//     Term 27 (APS4322-7000)/Term 28 (APS4322-5000)/FB Inputs/I{0..8 step 2} Y-Field <-> Data Pointer/HallSensorFieldsXYZ[{121..133 step 3}]  (5 links)
//     Term 27 (APS4322-7000)/Term 28 (APS4322-5000)/FB Inputs/I{0..8 step 2} Z-Field <-> Data Pointer/HallSensorFieldsXYZ[{122..134 step 3}]  (5 links)
//     Term 27 (APS4322-7000)/Term 28 (APS4322-5000)/FB Inputs/J{1..9 step 2} X-Field <-> Data Pointer/HallSensorFieldsXYZ[{135..147 step 3}]  (5 links)
//     Term 27 (APS4322-7000)/Term 28 (APS4322-5000)/FB Inputs/J{1..9 step 2} Y-Field <-> Data Pointer/HallSensorFieldsXYZ[{136..148 step 3}]  (5 links)
//     Term 27 (APS4322-7000)/Term 28 (APS4322-5000)/FB Inputs/J{1..9 step 2} Z-Field <-> Data Pointer/HallSensorFieldsXYZ[{137..149 step 3}]  (5 links)
//     Term 27 (APS4322-7000)/Term 28 (APS4322-5000)/FB Inputs/Status <-> Data Pointer/FeedbackStatus
//   Device 2 (EtherCAT) <-> TcCOM Objects/XPlanar/Part1/Tile3
//     Term 17 (APS4322-7000)/APS Comm Inputs/CommStatusWord <-> Data Pointer/MoverCommStatusWord
//     Term 17 (APS4322-7000)/APS Comm Inputs/Data {1..4} <-> Data Pointer/MoverCommDataIn[{0..3}]  (4 links)
//     Term 17 (APS4322-7000)/APS Comm Outputs/CommControlWord <-> Data Pointer/MoverCommControlWord
//     Term 17 (APS4322-7000)/APS Comm Outputs/Data 1 <-> Data Pointer/MoverCommDataOut
//     Term 17 (APS4322-7000)/APS Diagdata/DC Link Voltage <-> Data Pointer/DcLinkVoltage
//     Term 17 (APS4322-7000)/APS Diagdata/Power supply current <-> Data Pointer/PowerSupplyCurrent
//     Term 17 (APS4322-7000)/APS Inputs/StatusWord <-> Data Pointer/PowerUnitStatusWord
//     Term 17 (APS4322-7000)/APS Outputs/ControlWord <-> Data Pointer/PowerUnitControlWord
//     Term 17 (APS4322-7000)/APS Outputs/Current D 0X0 <-> Data Pointer/DCurrentSetPoints[0]
//     Term 17 (APS4322-7000)/APS Outputs/Current D 0X1 <-> Data Pointer/DCurrentSetPoints[1]
//     Term 17 (APS4322-7000)/APS Outputs/Current D 0X2 <-> Data Pointer/DCurrentSetPoints[2]
//     Term 17 (APS4322-7000)/APS Outputs/Current D 1X0 <-> Data Pointer/DCurrentSetPoints[6]
//     Term 17 (APS4322-7000)/APS Outputs/Current D 1X1 <-> Data Pointer/DCurrentSetPoints[7]
//     Term 17 (APS4322-7000)/APS Outputs/Current D 1X2 <-> Data Pointer/DCurrentSetPoints[8]
//     Term 17 (APS4322-7000)/APS Outputs/Current D 2X0 <-> Data Pointer/DCurrentSetPoints[12]
//     Term 17 (APS4322-7000)/APS Outputs/Current D 2X1 <-> Data Pointer/DCurrentSetPoints[13]
//     Term 17 (APS4322-7000)/APS Outputs/Current D 2X2 <-> Data Pointer/DCurrentSetPoints[14]
//     Term 17 (APS4322-7000)/APS Outputs/Current D 3X0 <-> Data Pointer/DCurrentSetPoints[18]
//     Term 17 (APS4322-7000)/APS Outputs/Current D 3X1 <-> Data Pointer/DCurrentSetPoints[19]
//     Term 17 (APS4322-7000)/APS Outputs/Current D 3X2 <-> Data Pointer/DCurrentSetPoints[20]
//     Term 17 (APS4322-7000)/APS Outputs/Current D 0Y0 <-> Data Pointer/DCurrentSetPoints[3]
//     Term 17 (APS4322-7000)/APS Outputs/Current D 0Y1 <-> Data Pointer/DCurrentSetPoints[4]
//     Term 17 (APS4322-7000)/APS Outputs/Current D 0Y2 <-> Data Pointer/DCurrentSetPoints[5]
//     Term 17 (APS4322-7000)/APS Outputs/Current D 1Y0 <-> Data Pointer/DCurrentSetPoints[9]
//     Term 17 (APS4322-7000)/APS Outputs/Current D 1Y1 <-> Data Pointer/DCurrentSetPoints[10]
//     Term 17 (APS4322-7000)/APS Outputs/Current D 1Y2 <-> Data Pointer/DCurrentSetPoints[11]
//     Term 17 (APS4322-7000)/APS Outputs/Current D 2Y0 <-> Data Pointer/DCurrentSetPoints[15]
//     Term 17 (APS4322-7000)/APS Outputs/Current D 2Y1 <-> Data Pointer/DCurrentSetPoints[16]
//     Term 17 (APS4322-7000)/APS Outputs/Current D 2Y2 <-> Data Pointer/DCurrentSetPoints[17]
//     Term 17 (APS4322-7000)/APS Outputs/Current D 3Y0 <-> Data Pointer/DCurrentSetPoints[21]
//     Term 17 (APS4322-7000)/APS Outputs/Current D 3Y1 <-> Data Pointer/DCurrentSetPoints[22]
//     Term 17 (APS4322-7000)/APS Outputs/Current D 3Y2 <-> Data Pointer/DCurrentSetPoints[23]
//     Term 17 (APS4322-7000)/APS Outputs/Current Q 0X0 <-> Data Pointer/QCurrentSetPoints[0]
//     Term 17 (APS4322-7000)/APS Outputs/Current Q 0X1 <-> Data Pointer/QCurrentSetPoints[1]
//     Term 17 (APS4322-7000)/APS Outputs/Current Q 0X2 <-> Data Pointer/QCurrentSetPoints[2]
//     Term 17 (APS4322-7000)/APS Outputs/Current Q 1X0 <-> Data Pointer/QCurrentSetPoints[6]
//     Term 17 (APS4322-7000)/APS Outputs/Current Q 1X1 <-> Data Pointer/QCurrentSetPoints[7]
//     Term 17 (APS4322-7000)/APS Outputs/Current Q 1X2 <-> Data Pointer/QCurrentSetPoints[8]
//     Term 17 (APS4322-7000)/APS Outputs/Current Q 2X0 <-> Data Pointer/QCurrentSetPoints[12]
//     Term 17 (APS4322-7000)/APS Outputs/Current Q 2X1 <-> Data Pointer/QCurrentSetPoints[13]
//     Term 17 (APS4322-7000)/APS Outputs/Current Q 2X2 <-> Data Pointer/QCurrentSetPoints[14]
//     Term 17 (APS4322-7000)/APS Outputs/Current Q 3X0 <-> Data Pointer/QCurrentSetPoints[18]
//     Term 17 (APS4322-7000)/APS Outputs/Current Q 3X1 <-> Data Pointer/QCurrentSetPoints[19]
//     Term 17 (APS4322-7000)/APS Outputs/Current Q 3X2 <-> Data Pointer/QCurrentSetPoints[20]
//     Term 17 (APS4322-7000)/APS Outputs/Current Q 0Y0 <-> Data Pointer/QCurrentSetPoints[3]
//     Term 17 (APS4322-7000)/APS Outputs/Current Q 0Y1 <-> Data Pointer/QCurrentSetPoints[4]
//     Term 17 (APS4322-7000)/APS Outputs/Current Q 0Y2 <-> Data Pointer/QCurrentSetPoints[5]
//     Term 17 (APS4322-7000)/APS Outputs/Current Q 1Y0 <-> Data Pointer/QCurrentSetPoints[9]
//     Term 17 (APS4322-7000)/APS Outputs/Current Q 1Y1 <-> Data Pointer/QCurrentSetPoints[10]
//     Term 17 (APS4322-7000)/APS Outputs/Current Q 1Y2 <-> Data Pointer/QCurrentSetPoints[11]
//     Term 17 (APS4322-7000)/APS Outputs/Current Q 2Y0 <-> Data Pointer/QCurrentSetPoints[15]
//     Term 17 (APS4322-7000)/APS Outputs/Current Q 2Y1 <-> Data Pointer/QCurrentSetPoints[16]
//     Term 17 (APS4322-7000)/APS Outputs/Current Q 2Y2 <-> Data Pointer/QCurrentSetPoints[17]
//     Term 17 (APS4322-7000)/APS Outputs/Current Q 3Y0 <-> Data Pointer/QCurrentSetPoints[21]
//     Term 17 (APS4322-7000)/APS Outputs/Current Q 3Y1 <-> Data Pointer/QCurrentSetPoints[22]
//     Term 17 (APS4322-7000)/APS Outputs/Current Q 3Y2 <-> Data Pointer/QCurrentSetPoints[23]
//     Term 17 (APS4322-7000)/APS Outputs/PhiE 0X0 <-> Data Pointer/PhiSetPoints[0]
//     Term 17 (APS4322-7000)/APS Outputs/PhiE 0X1 <-> Data Pointer/PhiSetPoints[1]
//     Term 17 (APS4322-7000)/APS Outputs/PhiE 0X2 <-> Data Pointer/PhiSetPoints[2]
//     Term 17 (APS4322-7000)/APS Outputs/PhiE 1X0 <-> Data Pointer/PhiSetPoints[6]
//     Term 17 (APS4322-7000)/APS Outputs/PhiE 1X1 <-> Data Pointer/PhiSetPoints[7]
//     Term 17 (APS4322-7000)/APS Outputs/PhiE 1X2 <-> Data Pointer/PhiSetPoints[8]
//     Term 17 (APS4322-7000)/APS Outputs/PhiE 2X0 <-> Data Pointer/PhiSetPoints[12]
//     Term 17 (APS4322-7000)/APS Outputs/PhiE 2X1 <-> Data Pointer/PhiSetPoints[13]
//     Term 17 (APS4322-7000)/APS Outputs/PhiE 2X2 <-> Data Pointer/PhiSetPoints[14]
//     Term 17 (APS4322-7000)/APS Outputs/PhiE 3X0 <-> Data Pointer/PhiSetPoints[18]
//     Term 17 (APS4322-7000)/APS Outputs/PhiE 3X1 <-> Data Pointer/PhiSetPoints[19]
//     Term 17 (APS4322-7000)/APS Outputs/PhiE 3X2 <-> Data Pointer/PhiSetPoints[20]
//     Term 17 (APS4322-7000)/APS Outputs/PhiE 0Y0 <-> Data Pointer/PhiSetPoints[3]
//     Term 17 (APS4322-7000)/APS Outputs/PhiE 0Y1 <-> Data Pointer/PhiSetPoints[4]
//     Term 17 (APS4322-7000)/APS Outputs/PhiE 0Y2 <-> Data Pointer/PhiSetPoints[5]
//     Term 17 (APS4322-7000)/APS Outputs/PhiE 1Y0 <-> Data Pointer/PhiSetPoints[9]
//     Term 17 (APS4322-7000)/APS Outputs/PhiE 1Y1 <-> Data Pointer/PhiSetPoints[10]
//     Term 17 (APS4322-7000)/APS Outputs/PhiE 1Y2 <-> Data Pointer/PhiSetPoints[11]
//     Term 17 (APS4322-7000)/APS Outputs/PhiE 2Y0 <-> Data Pointer/PhiSetPoints[15]
//     Term 17 (APS4322-7000)/APS Outputs/PhiE 2Y1 <-> Data Pointer/PhiSetPoints[16]
//     Term 17 (APS4322-7000)/APS Outputs/PhiE 2Y2 <-> Data Pointer/PhiSetPoints[17]
//     Term 17 (APS4322-7000)/APS Outputs/PhiE 3Y0 <-> Data Pointer/PhiSetPoints[21]
//     Term 17 (APS4322-7000)/APS Outputs/PhiE 3Y1 <-> Data Pointer/PhiSetPoints[22]
//     Term 17 (APS4322-7000)/APS Outputs/PhiE 3Y2 <-> Data Pointer/PhiSetPoints[23]
//     Term 17 (APS4322-7000)/Term 18 (APS4322-5000)/FB Inputs/A{0..8 step 2} X-Field <-> Data Pointer/HallSensorFieldsXYZ[{0..12 step 3}]  (5 links)
//     Term 17 (APS4322-7000)/Term 18 (APS4322-5000)/FB Inputs/A{0..8 step 2} Y-Field <-> Data Pointer/HallSensorFieldsXYZ[{1..13 step 3}]  (5 links)
//     Term 17 (APS4322-7000)/Term 18 (APS4322-5000)/FB Inputs/A{0..8 step 2} Z-Field <-> Data Pointer/HallSensorFieldsXYZ[{2..14 step 3}]  (5 links)
//     Term 17 (APS4322-7000)/Term 18 (APS4322-5000)/FB Inputs/B{1..9 step 2} X-Field <-> Data Pointer/HallSensorFieldsXYZ[{15..27 step 3}]  (5 links)
//     Term 17 (APS4322-7000)/Term 18 (APS4322-5000)/FB Inputs/B{1..9 step 2} Y-Field <-> Data Pointer/HallSensorFieldsXYZ[{16..28 step 3}]  (5 links)
//     Term 17 (APS4322-7000)/Term 18 (APS4322-5000)/FB Inputs/B{1..9 step 2} Z-Field <-> Data Pointer/HallSensorFieldsXYZ[{17..29 step 3}]  (5 links)
//     Term 17 (APS4322-7000)/Term 18 (APS4322-5000)/FB Inputs/C{0..8 step 2} X-Field <-> Data Pointer/HallSensorFieldsXYZ[{30..42 step 3}]  (5 links)
//     Term 17 (APS4322-7000)/Term 18 (APS4322-5000)/FB Inputs/C{0..8 step 2} Y-Field <-> Data Pointer/HallSensorFieldsXYZ[{31..43 step 3}]  (5 links)
//     Term 17 (APS4322-7000)/Term 18 (APS4322-5000)/FB Inputs/C{0..8 step 2} Z-Field <-> Data Pointer/HallSensorFieldsXYZ[{32..44 step 3}]  (5 links)
//     Term 17 (APS4322-7000)/Term 18 (APS4322-5000)/FB Inputs/D{1..9 step 2} X-Field <-> Data Pointer/HallSensorFieldsXYZ[{45..57 step 3}]  (5 links)
//     Term 17 (APS4322-7000)/Term 18 (APS4322-5000)/FB Inputs/D{1..9 step 2} Y-Field <-> Data Pointer/HallSensorFieldsXYZ[{46..58 step 3}]  (5 links)
//     Term 17 (APS4322-7000)/Term 18 (APS4322-5000)/FB Inputs/D{1..9 step 2} Z-Field <-> Data Pointer/HallSensorFieldsXYZ[{47..59 step 3}]  (5 links)
//     Term 17 (APS4322-7000)/Term 18 (APS4322-5000)/FB Inputs/E{0..8 step 2} X-Field <-> Data Pointer/HallSensorFieldsXYZ[{60..72 step 3}]  (5 links)
//     Term 17 (APS4322-7000)/Term 18 (APS4322-5000)/FB Inputs/E{0..8 step 2} Y-Field <-> Data Pointer/HallSensorFieldsXYZ[{61..73 step 3}]  (5 links)
//     Term 17 (APS4322-7000)/Term 18 (APS4322-5000)/FB Inputs/E{0..8 step 2} Z-Field <-> Data Pointer/HallSensorFieldsXYZ[{62..74 step 3}]  (5 links)
//     Term 17 (APS4322-7000)/Term 18 (APS4322-5000)/FB Inputs/F{1..9 step 2} X-Field <-> Data Pointer/HallSensorFieldsXYZ[{75..87 step 3}]  (5 links)
//     Term 17 (APS4322-7000)/Term 18 (APS4322-5000)/FB Inputs/F{1..9 step 2} Y-Field <-> Data Pointer/HallSensorFieldsXYZ[{76..88 step 3}]  (5 links)
//     Term 17 (APS4322-7000)/Term 18 (APS4322-5000)/FB Inputs/F{1..9 step 2} Z-Field <-> Data Pointer/HallSensorFieldsXYZ[{77..89 step 3}]  (5 links)
//     Term 17 (APS4322-7000)/Term 18 (APS4322-5000)/FB Inputs/G{0..8 step 2} X-Field <-> Data Pointer/HallSensorFieldsXYZ[{90..102 step 3}]  (5 links)
//     Term 17 (APS4322-7000)/Term 18 (APS4322-5000)/FB Inputs/G{0..8 step 2} Y-Field <-> Data Pointer/HallSensorFieldsXYZ[{91..103 step 3}]  (5 links)
//     Term 17 (APS4322-7000)/Term 18 (APS4322-5000)/FB Inputs/G{0..8 step 2} Z-Field <-> Data Pointer/HallSensorFieldsXYZ[{92..104 step 3}]  (5 links)
//     Term 17 (APS4322-7000)/Term 18 (APS4322-5000)/FB Inputs/H{1..9 step 2} X-Field <-> Data Pointer/HallSensorFieldsXYZ[{105..117 step 3}]  (5 links)
//     Term 17 (APS4322-7000)/Term 18 (APS4322-5000)/FB Inputs/H{1..9 step 2} Y-Field <-> Data Pointer/HallSensorFieldsXYZ[{106..118 step 3}]  (5 links)
//     Term 17 (APS4322-7000)/Term 18 (APS4322-5000)/FB Inputs/H{1..9 step 2} Z-Field <-> Data Pointer/HallSensorFieldsXYZ[{107..119 step 3}]  (5 links)
//     Term 17 (APS4322-7000)/Term 18 (APS4322-5000)/FB Inputs/I{0..8 step 2} X-Field <-> Data Pointer/HallSensorFieldsXYZ[{120..132 step 3}]  (5 links)
//     Term 17 (APS4322-7000)/Term 18 (APS4322-5000)/FB Inputs/I{0..8 step 2} Y-Field <-> Data Pointer/HallSensorFieldsXYZ[{121..133 step 3}]  (5 links)
//     Term 17 (APS4322-7000)/Term 18 (APS4322-5000)/FB Inputs/I{0..8 step 2} Z-Field <-> Data Pointer/HallSensorFieldsXYZ[{122..134 step 3}]  (5 links)
//     Term 17 (APS4322-7000)/Term 18 (APS4322-5000)/FB Inputs/J{1..9 step 2} X-Field <-> Data Pointer/HallSensorFieldsXYZ[{135..147 step 3}]  (5 links)
//     Term 17 (APS4322-7000)/Term 18 (APS4322-5000)/FB Inputs/J{1..9 step 2} Y-Field <-> Data Pointer/HallSensorFieldsXYZ[{136..148 step 3}]  (5 links)
//     Term 17 (APS4322-7000)/Term 18 (APS4322-5000)/FB Inputs/J{1..9 step 2} Z-Field <-> Data Pointer/HallSensorFieldsXYZ[{137..149 step 3}]  (5 links)
//     Term 17 (APS4322-7000)/Term 18 (APS4322-5000)/FB Inputs/Status <-> Data Pointer/FeedbackStatus
//   Device 2 (EtherCAT) <-> TcCOM Objects/XPlanar/Part1/Tile4
//     Term 19 (APS4322-7000)/APS Comm Inputs/CommStatusWord <-> Data Pointer/MoverCommStatusWord
//     Term 19 (APS4322-7000)/APS Comm Inputs/Data {1..4} <-> Data Pointer/MoverCommDataIn[{0..3}]  (4 links)
//     Term 19 (APS4322-7000)/APS Comm Outputs/CommControlWord <-> Data Pointer/MoverCommControlWord
//     Term 19 (APS4322-7000)/APS Comm Outputs/Data 1 <-> Data Pointer/MoverCommDataOut
//     Term 19 (APS4322-7000)/APS Diagdata/DC Link Voltage <-> Data Pointer/DcLinkVoltage
//     Term 19 (APS4322-7000)/APS Diagdata/Power supply current <-> Data Pointer/PowerSupplyCurrent
//     Term 19 (APS4322-7000)/APS Inputs/StatusWord <-> Data Pointer/PowerUnitStatusWord
//     Term 19 (APS4322-7000)/APS Outputs/ControlWord <-> Data Pointer/PowerUnitControlWord
//     Term 19 (APS4322-7000)/APS Outputs/Current D 0X0 <-> Data Pointer/DCurrentSetPoints[0]
//     Term 19 (APS4322-7000)/APS Outputs/Current D 0X1 <-> Data Pointer/DCurrentSetPoints[1]
//     Term 19 (APS4322-7000)/APS Outputs/Current D 0X2 <-> Data Pointer/DCurrentSetPoints[2]
//     Term 19 (APS4322-7000)/APS Outputs/Current D 1X0 <-> Data Pointer/DCurrentSetPoints[6]
//     Term 19 (APS4322-7000)/APS Outputs/Current D 1X1 <-> Data Pointer/DCurrentSetPoints[7]
//     Term 19 (APS4322-7000)/APS Outputs/Current D 1X2 <-> Data Pointer/DCurrentSetPoints[8]
//     Term 19 (APS4322-7000)/APS Outputs/Current D 2X0 <-> Data Pointer/DCurrentSetPoints[12]
//     Term 19 (APS4322-7000)/APS Outputs/Current D 2X1 <-> Data Pointer/DCurrentSetPoints[13]
//     Term 19 (APS4322-7000)/APS Outputs/Current D 2X2 <-> Data Pointer/DCurrentSetPoints[14]
//     Term 19 (APS4322-7000)/APS Outputs/Current D 3X0 <-> Data Pointer/DCurrentSetPoints[18]
//     Term 19 (APS4322-7000)/APS Outputs/Current D 3X1 <-> Data Pointer/DCurrentSetPoints[19]
//     Term 19 (APS4322-7000)/APS Outputs/Current D 3X2 <-> Data Pointer/DCurrentSetPoints[20]
//     Term 19 (APS4322-7000)/APS Outputs/Current D 0Y0 <-> Data Pointer/DCurrentSetPoints[3]
//     Term 19 (APS4322-7000)/APS Outputs/Current D 0Y1 <-> Data Pointer/DCurrentSetPoints[4]
//     Term 19 (APS4322-7000)/APS Outputs/Current D 0Y2 <-> Data Pointer/DCurrentSetPoints[5]
//     Term 19 (APS4322-7000)/APS Outputs/Current D 1Y0 <-> Data Pointer/DCurrentSetPoints[9]
//     Term 19 (APS4322-7000)/APS Outputs/Current D 1Y1 <-> Data Pointer/DCurrentSetPoints[10]
//     Term 19 (APS4322-7000)/APS Outputs/Current D 1Y2 <-> Data Pointer/DCurrentSetPoints[11]
//     Term 19 (APS4322-7000)/APS Outputs/Current D 2Y0 <-> Data Pointer/DCurrentSetPoints[15]
//     Term 19 (APS4322-7000)/APS Outputs/Current D 2Y1 <-> Data Pointer/DCurrentSetPoints[16]
//     Term 19 (APS4322-7000)/APS Outputs/Current D 2Y2 <-> Data Pointer/DCurrentSetPoints[17]
//     Term 19 (APS4322-7000)/APS Outputs/Current D 3Y0 <-> Data Pointer/DCurrentSetPoints[21]
//     Term 19 (APS4322-7000)/APS Outputs/Current D 3Y1 <-> Data Pointer/DCurrentSetPoints[22]
//     Term 19 (APS4322-7000)/APS Outputs/Current D 3Y2 <-> Data Pointer/DCurrentSetPoints[23]
//     Term 19 (APS4322-7000)/APS Outputs/Current Q 0X0 <-> Data Pointer/QCurrentSetPoints[0]
//     Term 19 (APS4322-7000)/APS Outputs/Current Q 0X1 <-> Data Pointer/QCurrentSetPoints[1]
//     Term 19 (APS4322-7000)/APS Outputs/Current Q 0X2 <-> Data Pointer/QCurrentSetPoints[2]
//     Term 19 (APS4322-7000)/APS Outputs/Current Q 1X0 <-> Data Pointer/QCurrentSetPoints[6]
//     Term 19 (APS4322-7000)/APS Outputs/Current Q 1X1 <-> Data Pointer/QCurrentSetPoints[7]
//     Term 19 (APS4322-7000)/APS Outputs/Current Q 1X2 <-> Data Pointer/QCurrentSetPoints[8]
//     Term 19 (APS4322-7000)/APS Outputs/Current Q 2X0 <-> Data Pointer/QCurrentSetPoints[12]
//     Term 19 (APS4322-7000)/APS Outputs/Current Q 2X1 <-> Data Pointer/QCurrentSetPoints[13]
//     Term 19 (APS4322-7000)/APS Outputs/Current Q 2X2 <-> Data Pointer/QCurrentSetPoints[14]
//     Term 19 (APS4322-7000)/APS Outputs/Current Q 3X0 <-> Data Pointer/QCurrentSetPoints[18]
//     Term 19 (APS4322-7000)/APS Outputs/Current Q 3X1 <-> Data Pointer/QCurrentSetPoints[19]
//     Term 19 (APS4322-7000)/APS Outputs/Current Q 3X2 <-> Data Pointer/QCurrentSetPoints[20]
//     Term 19 (APS4322-7000)/APS Outputs/Current Q 0Y0 <-> Data Pointer/QCurrentSetPoints[3]
//     Term 19 (APS4322-7000)/APS Outputs/Current Q 0Y1 <-> Data Pointer/QCurrentSetPoints[4]
//     Term 19 (APS4322-7000)/APS Outputs/Current Q 0Y2 <-> Data Pointer/QCurrentSetPoints[5]
//     Term 19 (APS4322-7000)/APS Outputs/Current Q 1Y0 <-> Data Pointer/QCurrentSetPoints[9]
//     Term 19 (APS4322-7000)/APS Outputs/Current Q 1Y1 <-> Data Pointer/QCurrentSetPoints[10]
//     Term 19 (APS4322-7000)/APS Outputs/Current Q 1Y2 <-> Data Pointer/QCurrentSetPoints[11]
//     Term 19 (APS4322-7000)/APS Outputs/Current Q 2Y0 <-> Data Pointer/QCurrentSetPoints[15]
//     Term 19 (APS4322-7000)/APS Outputs/Current Q 2Y1 <-> Data Pointer/QCurrentSetPoints[16]
//     Term 19 (APS4322-7000)/APS Outputs/Current Q 2Y2 <-> Data Pointer/QCurrentSetPoints[17]
//     Term 19 (APS4322-7000)/APS Outputs/Current Q 3Y0 <-> Data Pointer/QCurrentSetPoints[21]
//     Term 19 (APS4322-7000)/APS Outputs/Current Q 3Y1 <-> Data Pointer/QCurrentSetPoints[22]
//     Term 19 (APS4322-7000)/APS Outputs/Current Q 3Y2 <-> Data Pointer/QCurrentSetPoints[23]
//     Term 19 (APS4322-7000)/APS Outputs/PhiE 0X0 <-> Data Pointer/PhiSetPoints[0]
//     Term 19 (APS4322-7000)/APS Outputs/PhiE 0X1 <-> Data Pointer/PhiSetPoints[1]
//     Term 19 (APS4322-7000)/APS Outputs/PhiE 0X2 <-> Data Pointer/PhiSetPoints[2]
//     Term 19 (APS4322-7000)/APS Outputs/PhiE 1X0 <-> Data Pointer/PhiSetPoints[6]
//     Term 19 (APS4322-7000)/APS Outputs/PhiE 1X1 <-> Data Pointer/PhiSetPoints[7]
//     Term 19 (APS4322-7000)/APS Outputs/PhiE 1X2 <-> Data Pointer/PhiSetPoints[8]
//     Term 19 (APS4322-7000)/APS Outputs/PhiE 2X0 <-> Data Pointer/PhiSetPoints[12]
//     Term 19 (APS4322-7000)/APS Outputs/PhiE 2X1 <-> Data Pointer/PhiSetPoints[13]
//     Term 19 (APS4322-7000)/APS Outputs/PhiE 2X2 <-> Data Pointer/PhiSetPoints[14]
//     Term 19 (APS4322-7000)/APS Outputs/PhiE 3X0 <-> Data Pointer/PhiSetPoints[18]
//     Term 19 (APS4322-7000)/APS Outputs/PhiE 3X1 <-> Data Pointer/PhiSetPoints[19]
//     Term 19 (APS4322-7000)/APS Outputs/PhiE 3X2 <-> Data Pointer/PhiSetPoints[20]
//     Term 19 (APS4322-7000)/APS Outputs/PhiE 0Y0 <-> Data Pointer/PhiSetPoints[3]
//     Term 19 (APS4322-7000)/APS Outputs/PhiE 0Y1 <-> Data Pointer/PhiSetPoints[4]
//     Term 19 (APS4322-7000)/APS Outputs/PhiE 0Y2 <-> Data Pointer/PhiSetPoints[5]
//     Term 19 (APS4322-7000)/APS Outputs/PhiE 1Y0 <-> Data Pointer/PhiSetPoints[9]
//     Term 19 (APS4322-7000)/APS Outputs/PhiE 1Y1 <-> Data Pointer/PhiSetPoints[10]
//     Term 19 (APS4322-7000)/APS Outputs/PhiE 1Y2 <-> Data Pointer/PhiSetPoints[11]
//     Term 19 (APS4322-7000)/APS Outputs/PhiE 2Y0 <-> Data Pointer/PhiSetPoints[15]
//     Term 19 (APS4322-7000)/APS Outputs/PhiE 2Y1 <-> Data Pointer/PhiSetPoints[16]
//     Term 19 (APS4322-7000)/APS Outputs/PhiE 2Y2 <-> Data Pointer/PhiSetPoints[17]
//     Term 19 (APS4322-7000)/APS Outputs/PhiE 3Y0 <-> Data Pointer/PhiSetPoints[21]
//     Term 19 (APS4322-7000)/APS Outputs/PhiE 3Y1 <-> Data Pointer/PhiSetPoints[22]
//     Term 19 (APS4322-7000)/APS Outputs/PhiE 3Y2 <-> Data Pointer/PhiSetPoints[23]
//     Term 19 (APS4322-7000)/Term 20 (APS4322-5000)/FB Inputs/A{0..8 step 2} X-Field <-> Data Pointer/HallSensorFieldsXYZ[{0..12 step 3}]  (5 links)
//     Term 19 (APS4322-7000)/Term 20 (APS4322-5000)/FB Inputs/A{0..8 step 2} Y-Field <-> Data Pointer/HallSensorFieldsXYZ[{1..13 step 3}]  (5 links)
//     Term 19 (APS4322-7000)/Term 20 (APS4322-5000)/FB Inputs/A{0..8 step 2} Z-Field <-> Data Pointer/HallSensorFieldsXYZ[{2..14 step 3}]  (5 links)
//     Term 19 (APS4322-7000)/Term 20 (APS4322-5000)/FB Inputs/B{1..9 step 2} X-Field <-> Data Pointer/HallSensorFieldsXYZ[{15..27 step 3}]  (5 links)
//     Term 19 (APS4322-7000)/Term 20 (APS4322-5000)/FB Inputs/B{1..9 step 2} Y-Field <-> Data Pointer/HallSensorFieldsXYZ[{16..28 step 3}]  (5 links)
//     Term 19 (APS4322-7000)/Term 20 (APS4322-5000)/FB Inputs/B{1..9 step 2} Z-Field <-> Data Pointer/HallSensorFieldsXYZ[{17..29 step 3}]  (5 links)
//     Term 19 (APS4322-7000)/Term 20 (APS4322-5000)/FB Inputs/C{0..8 step 2} X-Field <-> Data Pointer/HallSensorFieldsXYZ[{30..42 step 3}]  (5 links)
//     Term 19 (APS4322-7000)/Term 20 (APS4322-5000)/FB Inputs/C{0..8 step 2} Y-Field <-> Data Pointer/HallSensorFieldsXYZ[{31..43 step 3}]  (5 links)
//     Term 19 (APS4322-7000)/Term 20 (APS4322-5000)/FB Inputs/C{0..8 step 2} Z-Field <-> Data Pointer/HallSensorFieldsXYZ[{32..44 step 3}]  (5 links)
//     Term 19 (APS4322-7000)/Term 20 (APS4322-5000)/FB Inputs/D{1..9 step 2} X-Field <-> Data Pointer/HallSensorFieldsXYZ[{45..57 step 3}]  (5 links)
//     Term 19 (APS4322-7000)/Term 20 (APS4322-5000)/FB Inputs/D{1..9 step 2} Y-Field <-> Data Pointer/HallSensorFieldsXYZ[{46..58 step 3}]  (5 links)
//     Term 19 (APS4322-7000)/Term 20 (APS4322-5000)/FB Inputs/D{1..9 step 2} Z-Field <-> Data Pointer/HallSensorFieldsXYZ[{47..59 step 3}]  (5 links)
//     Term 19 (APS4322-7000)/Term 20 (APS4322-5000)/FB Inputs/E{0..8 step 2} X-Field <-> Data Pointer/HallSensorFieldsXYZ[{60..72 step 3}]  (5 links)
//     Term 19 (APS4322-7000)/Term 20 (APS4322-5000)/FB Inputs/E{0..8 step 2} Y-Field <-> Data Pointer/HallSensorFieldsXYZ[{61..73 step 3}]  (5 links)
//     Term 19 (APS4322-7000)/Term 20 (APS4322-5000)/FB Inputs/E{0..8 step 2} Z-Field <-> Data Pointer/HallSensorFieldsXYZ[{62..74 step 3}]  (5 links)
//     Term 19 (APS4322-7000)/Term 20 (APS4322-5000)/FB Inputs/F{1..9 step 2} X-Field <-> Data Pointer/HallSensorFieldsXYZ[{75..87 step 3}]  (5 links)
//     Term 19 (APS4322-7000)/Term 20 (APS4322-5000)/FB Inputs/F{1..9 step 2} Y-Field <-> Data Pointer/HallSensorFieldsXYZ[{76..88 step 3}]  (5 links)
//     Term 19 (APS4322-7000)/Term 20 (APS4322-5000)/FB Inputs/F{1..9 step 2} Z-Field <-> Data Pointer/HallSensorFieldsXYZ[{77..89 step 3}]  (5 links)
//     Term 19 (APS4322-7000)/Term 20 (APS4322-5000)/FB Inputs/G{0..8 step 2} X-Field <-> Data Pointer/HallSensorFieldsXYZ[{90..102 step 3}]  (5 links)
//     Term 19 (APS4322-7000)/Term 20 (APS4322-5000)/FB Inputs/G{0..8 step 2} Y-Field <-> Data Pointer/HallSensorFieldsXYZ[{91..103 step 3}]  (5 links)
//     Term 19 (APS4322-7000)/Term 20 (APS4322-5000)/FB Inputs/G{0..8 step 2} Z-Field <-> Data Pointer/HallSensorFieldsXYZ[{92..104 step 3}]  (5 links)
//     Term 19 (APS4322-7000)/Term 20 (APS4322-5000)/FB Inputs/H{1..9 step 2} X-Field <-> Data Pointer/HallSensorFieldsXYZ[{105..117 step 3}]  (5 links)
//     Term 19 (APS4322-7000)/Term 20 (APS4322-5000)/FB Inputs/H{1..9 step 2} Y-Field <-> Data Pointer/HallSensorFieldsXYZ[{106..118 step 3}]  (5 links)
//     Term 19 (APS4322-7000)/Term 20 (APS4322-5000)/FB Inputs/H{1..9 step 2} Z-Field <-> Data Pointer/HallSensorFieldsXYZ[{107..119 step 3}]  (5 links)
//     Term 19 (APS4322-7000)/Term 20 (APS4322-5000)/FB Inputs/I{0..8 step 2} X-Field <-> Data Pointer/HallSensorFieldsXYZ[{120..132 step 3}]  (5 links)
//     Term 19 (APS4322-7000)/Term 20 (APS4322-5000)/FB Inputs/I{0..8 step 2} Y-Field <-> Data Pointer/HallSensorFieldsXYZ[{121..133 step 3}]  (5 links)
//     Term 19 (APS4322-7000)/Term 20 (APS4322-5000)/FB Inputs/I{0..8 step 2} Z-Field <-> Data Pointer/HallSensorFieldsXYZ[{122..134 step 3}]  (5 links)
//     Term 19 (APS4322-7000)/Term 20 (APS4322-5000)/FB Inputs/J{1..9 step 2} X-Field <-> Data Pointer/HallSensorFieldsXYZ[{135..147 step 3}]  (5 links)
//     Term 19 (APS4322-7000)/Term 20 (APS4322-5000)/FB Inputs/J{1..9 step 2} Y-Field <-> Data Pointer/HallSensorFieldsXYZ[{136..148 step 3}]  (5 links)
//     Term 19 (APS4322-7000)/Term 20 (APS4322-5000)/FB Inputs/J{1..9 step 2} Z-Field <-> Data Pointer/HallSensorFieldsXYZ[{137..149 step 3}]  (5 links)
//     Term 19 (APS4322-7000)/Term 20 (APS4322-5000)/FB Inputs/Status <-> Data Pointer/FeedbackStatus
//   Device 2 (EtherCAT) <-> TcCOM Objects/XPlanar/Part1/Tile7
//     Term 21 (APS4322-7000)/APS Comm Inputs/CommStatusWord <-> Data Pointer/MoverCommStatusWord
//     Term 21 (APS4322-7000)/APS Comm Inputs/Data {1..4} <-> Data Pointer/MoverCommDataIn[{0..3}]  (4 links)
//     Term 21 (APS4322-7000)/APS Comm Outputs/CommControlWord <-> Data Pointer/MoverCommControlWord
//     Term 21 (APS4322-7000)/APS Comm Outputs/Data 1 <-> Data Pointer/MoverCommDataOut
//     Term 21 (APS4322-7000)/APS Diagdata/DC Link Voltage <-> Data Pointer/DcLinkVoltage
//     Term 21 (APS4322-7000)/APS Diagdata/Power supply current <-> Data Pointer/PowerSupplyCurrent
//     Term 21 (APS4322-7000)/APS Inputs/StatusWord <-> Data Pointer/PowerUnitStatusWord
//     Term 21 (APS4322-7000)/APS Outputs/ControlWord <-> Data Pointer/PowerUnitControlWord
//     Term 21 (APS4322-7000)/APS Outputs/Current D 0X0 <-> Data Pointer/DCurrentSetPoints[0]
//     Term 21 (APS4322-7000)/APS Outputs/Current D 0X1 <-> Data Pointer/DCurrentSetPoints[1]
//     Term 21 (APS4322-7000)/APS Outputs/Current D 0X2 <-> Data Pointer/DCurrentSetPoints[2]
//     Term 21 (APS4322-7000)/APS Outputs/Current D 1X0 <-> Data Pointer/DCurrentSetPoints[6]
//     Term 21 (APS4322-7000)/APS Outputs/Current D 1X1 <-> Data Pointer/DCurrentSetPoints[7]
//     Term 21 (APS4322-7000)/APS Outputs/Current D 1X2 <-> Data Pointer/DCurrentSetPoints[8]
//     Term 21 (APS4322-7000)/APS Outputs/Current D 2X0 <-> Data Pointer/DCurrentSetPoints[12]
//     Term 21 (APS4322-7000)/APS Outputs/Current D 2X1 <-> Data Pointer/DCurrentSetPoints[13]
//     Term 21 (APS4322-7000)/APS Outputs/Current D 2X2 <-> Data Pointer/DCurrentSetPoints[14]
//     Term 21 (APS4322-7000)/APS Outputs/Current D 3X0 <-> Data Pointer/DCurrentSetPoints[18]
//     Term 21 (APS4322-7000)/APS Outputs/Current D 3X1 <-> Data Pointer/DCurrentSetPoints[19]
//     Term 21 (APS4322-7000)/APS Outputs/Current D 3X2 <-> Data Pointer/DCurrentSetPoints[20]
//     Term 21 (APS4322-7000)/APS Outputs/Current D 0Y0 <-> Data Pointer/DCurrentSetPoints[3]
//     Term 21 (APS4322-7000)/APS Outputs/Current D 0Y1 <-> Data Pointer/DCurrentSetPoints[4]
//     Term 21 (APS4322-7000)/APS Outputs/Current D 0Y2 <-> Data Pointer/DCurrentSetPoints[5]
//     Term 21 (APS4322-7000)/APS Outputs/Current D 1Y0 <-> Data Pointer/DCurrentSetPoints[9]
//     Term 21 (APS4322-7000)/APS Outputs/Current D 1Y1 <-> Data Pointer/DCurrentSetPoints[10]
//     Term 21 (APS4322-7000)/APS Outputs/Current D 1Y2 <-> Data Pointer/DCurrentSetPoints[11]
//     Term 21 (APS4322-7000)/APS Outputs/Current D 2Y0 <-> Data Pointer/DCurrentSetPoints[15]
//     Term 21 (APS4322-7000)/APS Outputs/Current D 2Y1 <-> Data Pointer/DCurrentSetPoints[16]
//     Term 21 (APS4322-7000)/APS Outputs/Current D 2Y2 <-> Data Pointer/DCurrentSetPoints[17]
//     Term 21 (APS4322-7000)/APS Outputs/Current D 3Y0 <-> Data Pointer/DCurrentSetPoints[21]
//     Term 21 (APS4322-7000)/APS Outputs/Current D 3Y1 <-> Data Pointer/DCurrentSetPoints[22]
//     Term 21 (APS4322-7000)/APS Outputs/Current D 3Y2 <-> Data Pointer/DCurrentSetPoints[23]
//     Term 21 (APS4322-7000)/APS Outputs/Current Q 0X0 <-> Data Pointer/QCurrentSetPoints[0]
//     Term 21 (APS4322-7000)/APS Outputs/Current Q 0X1 <-> Data Pointer/QCurrentSetPoints[1]
//     Term 21 (APS4322-7000)/APS Outputs/Current Q 0X2 <-> Data Pointer/QCurrentSetPoints[2]
//     Term 21 (APS4322-7000)/APS Outputs/Current Q 1X0 <-> Data Pointer/QCurrentSetPoints[6]
//     Term 21 (APS4322-7000)/APS Outputs/Current Q 1X1 <-> Data Pointer/QCurrentSetPoints[7]
//     Term 21 (APS4322-7000)/APS Outputs/Current Q 1X2 <-> Data Pointer/QCurrentSetPoints[8]
//     Term 21 (APS4322-7000)/APS Outputs/Current Q 2X0 <-> Data Pointer/QCurrentSetPoints[12]
//     Term 21 (APS4322-7000)/APS Outputs/Current Q 2X1 <-> Data Pointer/QCurrentSetPoints[13]
//     Term 21 (APS4322-7000)/APS Outputs/Current Q 2X2 <-> Data Pointer/QCurrentSetPoints[14]
//     Term 21 (APS4322-7000)/APS Outputs/Current Q 3X0 <-> Data Pointer/QCurrentSetPoints[18]
//     Term 21 (APS4322-7000)/APS Outputs/Current Q 3X1 <-> Data Pointer/QCurrentSetPoints[19]
//     Term 21 (APS4322-7000)/APS Outputs/Current Q 3X2 <-> Data Pointer/QCurrentSetPoints[20]
//     Term 21 (APS4322-7000)/APS Outputs/Current Q 0Y0 <-> Data Pointer/QCurrentSetPoints[3]
//     Term 21 (APS4322-7000)/APS Outputs/Current Q 0Y1 <-> Data Pointer/QCurrentSetPoints[4]
//     Term 21 (APS4322-7000)/APS Outputs/Current Q 0Y2 <-> Data Pointer/QCurrentSetPoints[5]
//     Term 21 (APS4322-7000)/APS Outputs/Current Q 1Y0 <-> Data Pointer/QCurrentSetPoints[9]
//     Term 21 (APS4322-7000)/APS Outputs/Current Q 1Y1 <-> Data Pointer/QCurrentSetPoints[10]
//     Term 21 (APS4322-7000)/APS Outputs/Current Q 1Y2 <-> Data Pointer/QCurrentSetPoints[11]
//     Term 21 (APS4322-7000)/APS Outputs/Current Q 2Y0 <-> Data Pointer/QCurrentSetPoints[15]
//     Term 21 (APS4322-7000)/APS Outputs/Current Q 2Y1 <-> Data Pointer/QCurrentSetPoints[16]
//     Term 21 (APS4322-7000)/APS Outputs/Current Q 2Y2 <-> Data Pointer/QCurrentSetPoints[17]
//     Term 21 (APS4322-7000)/APS Outputs/Current Q 3Y0 <-> Data Pointer/QCurrentSetPoints[21]
//     Term 21 (APS4322-7000)/APS Outputs/Current Q 3Y1 <-> Data Pointer/QCurrentSetPoints[22]
//     Term 21 (APS4322-7000)/APS Outputs/Current Q 3Y2 <-> Data Pointer/QCurrentSetPoints[23]
//     Term 21 (APS4322-7000)/APS Outputs/PhiE 0X0 <-> Data Pointer/PhiSetPoints[0]
//     Term 21 (APS4322-7000)/APS Outputs/PhiE 0X1 <-> Data Pointer/PhiSetPoints[1]
//     Term 21 (APS4322-7000)/APS Outputs/PhiE 0X2 <-> Data Pointer/PhiSetPoints[2]
//     Term 21 (APS4322-7000)/APS Outputs/PhiE 1X0 <-> Data Pointer/PhiSetPoints[6]
//     Term 21 (APS4322-7000)/APS Outputs/PhiE 1X1 <-> Data Pointer/PhiSetPoints[7]
//     Term 21 (APS4322-7000)/APS Outputs/PhiE 1X2 <-> Data Pointer/PhiSetPoints[8]
//     Term 21 (APS4322-7000)/APS Outputs/PhiE 2X0 <-> Data Pointer/PhiSetPoints[12]
//     Term 21 (APS4322-7000)/APS Outputs/PhiE 2X1 <-> Data Pointer/PhiSetPoints[13]
//     Term 21 (APS4322-7000)/APS Outputs/PhiE 2X2 <-> Data Pointer/PhiSetPoints[14]
//     Term 21 (APS4322-7000)/APS Outputs/PhiE 3X0 <-> Data Pointer/PhiSetPoints[18]
//     Term 21 (APS4322-7000)/APS Outputs/PhiE 3X1 <-> Data Pointer/PhiSetPoints[19]
//     Term 21 (APS4322-7000)/APS Outputs/PhiE 3X2 <-> Data Pointer/PhiSetPoints[20]
//     Term 21 (APS4322-7000)/APS Outputs/PhiE 0Y0 <-> Data Pointer/PhiSetPoints[3]
//     Term 21 (APS4322-7000)/APS Outputs/PhiE 0Y1 <-> Data Pointer/PhiSetPoints[4]
//     Term 21 (APS4322-7000)/APS Outputs/PhiE 0Y2 <-> Data Pointer/PhiSetPoints[5]
//     Term 21 (APS4322-7000)/APS Outputs/PhiE 1Y0 <-> Data Pointer/PhiSetPoints[9]
//     Term 21 (APS4322-7000)/APS Outputs/PhiE 1Y1 <-> Data Pointer/PhiSetPoints[10]
//     Term 21 (APS4322-7000)/APS Outputs/PhiE 1Y2 <-> Data Pointer/PhiSetPoints[11]
//     Term 21 (APS4322-7000)/APS Outputs/PhiE 2Y0 <-> Data Pointer/PhiSetPoints[15]
//     Term 21 (APS4322-7000)/APS Outputs/PhiE 2Y1 <-> Data Pointer/PhiSetPoints[16]
//     Term 21 (APS4322-7000)/APS Outputs/PhiE 2Y2 <-> Data Pointer/PhiSetPoints[17]
//     Term 21 (APS4322-7000)/APS Outputs/PhiE 3Y0 <-> Data Pointer/PhiSetPoints[21]
//     Term 21 (APS4322-7000)/APS Outputs/PhiE 3Y1 <-> Data Pointer/PhiSetPoints[22]
//     Term 21 (APS4322-7000)/APS Outputs/PhiE 3Y2 <-> Data Pointer/PhiSetPoints[23]
//     Term 21 (APS4322-7000)/Term 22 (APS4322-5000)/FB Inputs/A{0..8 step 2} X-Field <-> Data Pointer/HallSensorFieldsXYZ[{0..12 step 3}]  (5 links)
//     Term 21 (APS4322-7000)/Term 22 (APS4322-5000)/FB Inputs/A{0..8 step 2} Y-Field <-> Data Pointer/HallSensorFieldsXYZ[{1..13 step 3}]  (5 links)
//     Term 21 (APS4322-7000)/Term 22 (APS4322-5000)/FB Inputs/A{0..8 step 2} Z-Field <-> Data Pointer/HallSensorFieldsXYZ[{2..14 step 3}]  (5 links)
//     Term 21 (APS4322-7000)/Term 22 (APS4322-5000)/FB Inputs/B{1..9 step 2} X-Field <-> Data Pointer/HallSensorFieldsXYZ[{15..27 step 3}]  (5 links)
//     Term 21 (APS4322-7000)/Term 22 (APS4322-5000)/FB Inputs/B{1..9 step 2} Y-Field <-> Data Pointer/HallSensorFieldsXYZ[{16..28 step 3}]  (5 links)
//     Term 21 (APS4322-7000)/Term 22 (APS4322-5000)/FB Inputs/B{1..9 step 2} Z-Field <-> Data Pointer/HallSensorFieldsXYZ[{17..29 step 3}]  (5 links)
//     Term 21 (APS4322-7000)/Term 22 (APS4322-5000)/FB Inputs/C{0..8 step 2} X-Field <-> Data Pointer/HallSensorFieldsXYZ[{30..42 step 3}]  (5 links)
//     Term 21 (APS4322-7000)/Term 22 (APS4322-5000)/FB Inputs/C{0..8 step 2} Y-Field <-> Data Pointer/HallSensorFieldsXYZ[{31..43 step 3}]  (5 links)
//     Term 21 (APS4322-7000)/Term 22 (APS4322-5000)/FB Inputs/C{0..8 step 2} Z-Field <-> Data Pointer/HallSensorFieldsXYZ[{32..44 step 3}]  (5 links)
//     Term 21 (APS4322-7000)/Term 22 (APS4322-5000)/FB Inputs/D{1..9 step 2} X-Field <-> Data Pointer/HallSensorFieldsXYZ[{45..57 step 3}]  (5 links)
//     Term 21 (APS4322-7000)/Term 22 (APS4322-5000)/FB Inputs/D{1..9 step 2} Y-Field <-> Data Pointer/HallSensorFieldsXYZ[{46..58 step 3}]  (5 links)
//     Term 21 (APS4322-7000)/Term 22 (APS4322-5000)/FB Inputs/D{1..9 step 2} Z-Field <-> Data Pointer/HallSensorFieldsXYZ[{47..59 step 3}]  (5 links)
//     Term 21 (APS4322-7000)/Term 22 (APS4322-5000)/FB Inputs/E{0..8 step 2} X-Field <-> Data Pointer/HallSensorFieldsXYZ[{60..72 step 3}]  (5 links)
//     Term 21 (APS4322-7000)/Term 22 (APS4322-5000)/FB Inputs/E{0..8 step 2} Y-Field <-> Data Pointer/HallSensorFieldsXYZ[{61..73 step 3}]  (5 links)
//     Term 21 (APS4322-7000)/Term 22 (APS4322-5000)/FB Inputs/E{0..8 step 2} Z-Field <-> Data Pointer/HallSensorFieldsXYZ[{62..74 step 3}]  (5 links)
//     Term 21 (APS4322-7000)/Term 22 (APS4322-5000)/FB Inputs/F{1..9 step 2} X-Field <-> Data Pointer/HallSensorFieldsXYZ[{75..87 step 3}]  (5 links)
//     Term 21 (APS4322-7000)/Term 22 (APS4322-5000)/FB Inputs/F{1..9 step 2} Y-Field <-> Data Pointer/HallSensorFieldsXYZ[{76..88 step 3}]  (5 links)
//     Term 21 (APS4322-7000)/Term 22 (APS4322-5000)/FB Inputs/F{1..9 step 2} Z-Field <-> Data Pointer/HallSensorFieldsXYZ[{77..89 step 3}]  (5 links)
//     Term 21 (APS4322-7000)/Term 22 (APS4322-5000)/FB Inputs/G{0..8 step 2} X-Field <-> Data Pointer/HallSensorFieldsXYZ[{90..102 step 3}]  (5 links)
//     Term 21 (APS4322-7000)/Term 22 (APS4322-5000)/FB Inputs/G{0..8 step 2} Y-Field <-> Data Pointer/HallSensorFieldsXYZ[{91..103 step 3}]  (5 links)
//     Term 21 (APS4322-7000)/Term 22 (APS4322-5000)/FB Inputs/G{0..8 step 2} Z-Field <-> Data Pointer/HallSensorFieldsXYZ[{92..104 step 3}]  (5 links)
//     Term 21 (APS4322-7000)/Term 22 (APS4322-5000)/FB Inputs/H{1..9 step 2} X-Field <-> Data Pointer/HallSensorFieldsXYZ[{105..117 step 3}]  (5 links)
//     Term 21 (APS4322-7000)/Term 22 (APS4322-5000)/FB Inputs/H{1..9 step 2} Y-Field <-> Data Pointer/HallSensorFieldsXYZ[{106..118 step 3}]  (5 links)
//     Term 21 (APS4322-7000)/Term 22 (APS4322-5000)/FB Inputs/H{1..9 step 2} Z-Field <-> Data Pointer/HallSensorFieldsXYZ[{107..119 step 3}]  (5 links)
//     Term 21 (APS4322-7000)/Term 22 (APS4322-5000)/FB Inputs/I{0..8 step 2} X-Field <-> Data Pointer/HallSensorFieldsXYZ[{120..132 step 3}]  (5 links)
//     Term 21 (APS4322-7000)/Term 22 (APS4322-5000)/FB Inputs/I{0..8 step 2} Y-Field <-> Data Pointer/HallSensorFieldsXYZ[{121..133 step 3}]  (5 links)
//     Term 21 (APS4322-7000)/Term 22 (APS4322-5000)/FB Inputs/I{0..8 step 2} Z-Field <-> Data Pointer/HallSensorFieldsXYZ[{122..134 step 3}]  (5 links)
//     Term 21 (APS4322-7000)/Term 22 (APS4322-5000)/FB Inputs/J{1..9 step 2} X-Field <-> Data Pointer/HallSensorFieldsXYZ[{135..147 step 3}]  (5 links)
//     Term 21 (APS4322-7000)/Term 22 (APS4322-5000)/FB Inputs/J{1..9 step 2} Y-Field <-> Data Pointer/HallSensorFieldsXYZ[{136..148 step 3}]  (5 links)
//     Term 21 (APS4322-7000)/Term 22 (APS4322-5000)/FB Inputs/J{1..9 step 2} Z-Field <-> Data Pointer/HallSensorFieldsXYZ[{137..149 step 3}]  (5 links)
//     Term 21 (APS4322-7000)/Term 22 (APS4322-5000)/FB Inputs/Status <-> Data Pointer/FeedbackStatus
//   Device 2 (EtherCAT) <-> TcCOM Objects/XPlanar/Part1/Tile8
//     Term 23 (APS4322-7000)/APS Comm Inputs/CommStatusWord <-> Data Pointer/MoverCommStatusWord
//     Term 23 (APS4322-7000)/APS Comm Inputs/Data {1..4} <-> Data Pointer/MoverCommDataIn[{0..3}]  (4 links)
//     Term 23 (APS4322-7000)/APS Comm Outputs/CommControlWord <-> Data Pointer/MoverCommControlWord
//     Term 23 (APS4322-7000)/APS Comm Outputs/Data 1 <-> Data Pointer/MoverCommDataOut
//     Term 23 (APS4322-7000)/APS Diagdata/DC Link Voltage <-> Data Pointer/DcLinkVoltage
//     Term 23 (APS4322-7000)/APS Diagdata/Power supply current <-> Data Pointer/PowerSupplyCurrent
//     Term 23 (APS4322-7000)/APS Inputs/StatusWord <-> Data Pointer/PowerUnitStatusWord
//     Term 23 (APS4322-7000)/APS Outputs/ControlWord <-> Data Pointer/PowerUnitControlWord
//     Term 23 (APS4322-7000)/APS Outputs/Current D 0X0 <-> Data Pointer/DCurrentSetPoints[0]
//     Term 23 (APS4322-7000)/APS Outputs/Current D 0X1 <-> Data Pointer/DCurrentSetPoints[1]
//     Term 23 (APS4322-7000)/APS Outputs/Current D 0X2 <-> Data Pointer/DCurrentSetPoints[2]
//     Term 23 (APS4322-7000)/APS Outputs/Current D 1X0 <-> Data Pointer/DCurrentSetPoints[6]
//     Term 23 (APS4322-7000)/APS Outputs/Current D 1X1 <-> Data Pointer/DCurrentSetPoints[7]
//     Term 23 (APS4322-7000)/APS Outputs/Current D 1X2 <-> Data Pointer/DCurrentSetPoints[8]
//     Term 23 (APS4322-7000)/APS Outputs/Current D 2X0 <-> Data Pointer/DCurrentSetPoints[12]
//     Term 23 (APS4322-7000)/APS Outputs/Current D 2X1 <-> Data Pointer/DCurrentSetPoints[13]
//     Term 23 (APS4322-7000)/APS Outputs/Current D 2X2 <-> Data Pointer/DCurrentSetPoints[14]
//     Term 23 (APS4322-7000)/APS Outputs/Current D 3X0 <-> Data Pointer/DCurrentSetPoints[18]
//     Term 23 (APS4322-7000)/APS Outputs/Current D 3X1 <-> Data Pointer/DCurrentSetPoints[19]
//     Term 23 (APS4322-7000)/APS Outputs/Current D 3X2 <-> Data Pointer/DCurrentSetPoints[20]
//     Term 23 (APS4322-7000)/APS Outputs/Current D 0Y0 <-> Data Pointer/DCurrentSetPoints[3]
//     Term 23 (APS4322-7000)/APS Outputs/Current D 0Y1 <-> Data Pointer/DCurrentSetPoints[4]
//     Term 23 (APS4322-7000)/APS Outputs/Current D 0Y2 <-> Data Pointer/DCurrentSetPoints[5]
//     Term 23 (APS4322-7000)/APS Outputs/Current D 1Y0 <-> Data Pointer/DCurrentSetPoints[9]
//     Term 23 (APS4322-7000)/APS Outputs/Current D 1Y1 <-> Data Pointer/DCurrentSetPoints[10]
//     Term 23 (APS4322-7000)/APS Outputs/Current D 1Y2 <-> Data Pointer/DCurrentSetPoints[11]
//     Term 23 (APS4322-7000)/APS Outputs/Current D 2Y0 <-> Data Pointer/DCurrentSetPoints[15]
//     Term 23 (APS4322-7000)/APS Outputs/Current D 2Y1 <-> Data Pointer/DCurrentSetPoints[16]
//     Term 23 (APS4322-7000)/APS Outputs/Current D 2Y2 <-> Data Pointer/DCurrentSetPoints[17]
//     Term 23 (APS4322-7000)/APS Outputs/Current D 3Y0 <-> Data Pointer/DCurrentSetPoints[21]
//     Term 23 (APS4322-7000)/APS Outputs/Current D 3Y1 <-> Data Pointer/DCurrentSetPoints[22]
//     Term 23 (APS4322-7000)/APS Outputs/Current D 3Y2 <-> Data Pointer/DCurrentSetPoints[23]
//     Term 23 (APS4322-7000)/APS Outputs/Current Q 0X0 <-> Data Pointer/QCurrentSetPoints[0]
//     Term 23 (APS4322-7000)/APS Outputs/Current Q 0X1 <-> Data Pointer/QCurrentSetPoints[1]
//     Term 23 (APS4322-7000)/APS Outputs/Current Q 0X2 <-> Data Pointer/QCurrentSetPoints[2]
//     Term 23 (APS4322-7000)/APS Outputs/Current Q 1X0 <-> Data Pointer/QCurrentSetPoints[6]
//     Term 23 (APS4322-7000)/APS Outputs/Current Q 1X1 <-> Data Pointer/QCurrentSetPoints[7]
//     Term 23 (APS4322-7000)/APS Outputs/Current Q 1X2 <-> Data Pointer/QCurrentSetPoints[8]
//     Term 23 (APS4322-7000)/APS Outputs/Current Q 2X0 <-> Data Pointer/QCurrentSetPoints[12]
//     Term 23 (APS4322-7000)/APS Outputs/Current Q 2X1 <-> Data Pointer/QCurrentSetPoints[13]
//     Term 23 (APS4322-7000)/APS Outputs/Current Q 2X2 <-> Data Pointer/QCurrentSetPoints[14]
//     Term 23 (APS4322-7000)/APS Outputs/Current Q 3X0 <-> Data Pointer/QCurrentSetPoints[18]
//     Term 23 (APS4322-7000)/APS Outputs/Current Q 3X1 <-> Data Pointer/QCurrentSetPoints[19]
//     Term 23 (APS4322-7000)/APS Outputs/Current Q 3X2 <-> Data Pointer/QCurrentSetPoints[20]
//     Term 23 (APS4322-7000)/APS Outputs/Current Q 0Y0 <-> Data Pointer/QCurrentSetPoints[3]
//     Term 23 (APS4322-7000)/APS Outputs/Current Q 0Y1 <-> Data Pointer/QCurrentSetPoints[4]
//     Term 23 (APS4322-7000)/APS Outputs/Current Q 0Y2 <-> Data Pointer/QCurrentSetPoints[5]
//     Term 23 (APS4322-7000)/APS Outputs/Current Q 1Y0 <-> Data Pointer/QCurrentSetPoints[9]
//     Term 23 (APS4322-7000)/APS Outputs/Current Q 1Y1 <-> Data Pointer/QCurrentSetPoints[10]
//     Term 23 (APS4322-7000)/APS Outputs/Current Q 1Y2 <-> Data Pointer/QCurrentSetPoints[11]
//     Term 23 (APS4322-7000)/APS Outputs/Current Q 2Y0 <-> Data Pointer/QCurrentSetPoints[15]
//     Term 23 (APS4322-7000)/APS Outputs/Current Q 2Y1 <-> Data Pointer/QCurrentSetPoints[16]
//     Term 23 (APS4322-7000)/APS Outputs/Current Q 2Y2 <-> Data Pointer/QCurrentSetPoints[17]
//     Term 23 (APS4322-7000)/APS Outputs/Current Q 3Y0 <-> Data Pointer/QCurrentSetPoints[21]
//     Term 23 (APS4322-7000)/APS Outputs/Current Q 3Y1 <-> Data Pointer/QCurrentSetPoints[22]
//     Term 23 (APS4322-7000)/APS Outputs/Current Q 3Y2 <-> Data Pointer/QCurrentSetPoints[23]
//     Term 23 (APS4322-7000)/APS Outputs/PhiE 0X0 <-> Data Pointer/PhiSetPoints[0]
//     Term 23 (APS4322-7000)/APS Outputs/PhiE 0X1 <-> Data Pointer/PhiSetPoints[1]
//     Term 23 (APS4322-7000)/APS Outputs/PhiE 0X2 <-> Data Pointer/PhiSetPoints[2]
//     Term 23 (APS4322-7000)/APS Outputs/PhiE 1X0 <-> Data Pointer/PhiSetPoints[6]
//     Term 23 (APS4322-7000)/APS Outputs/PhiE 1X1 <-> Data Pointer/PhiSetPoints[7]
//     Term 23 (APS4322-7000)/APS Outputs/PhiE 1X2 <-> Data Pointer/PhiSetPoints[8]
//     Term 23 (APS4322-7000)/APS Outputs/PhiE 2X0 <-> Data Pointer/PhiSetPoints[12]
//     Term 23 (APS4322-7000)/APS Outputs/PhiE 2X1 <-> Data Pointer/PhiSetPoints[13]
//     Term 23 (APS4322-7000)/APS Outputs/PhiE 2X2 <-> Data Pointer/PhiSetPoints[14]
//     Term 23 (APS4322-7000)/APS Outputs/PhiE 3X0 <-> Data Pointer/PhiSetPoints[18]
//     Term 23 (APS4322-7000)/APS Outputs/PhiE 3X1 <-> Data Pointer/PhiSetPoints[19]
//     Term 23 (APS4322-7000)/APS Outputs/PhiE 3X2 <-> Data Pointer/PhiSetPoints[20]
//     Term 23 (APS4322-7000)/APS Outputs/PhiE 0Y0 <-> Data Pointer/PhiSetPoints[3]
//     Term 23 (APS4322-7000)/APS Outputs/PhiE 0Y1 <-> Data Pointer/PhiSetPoints[4]
//     Term 23 (APS4322-7000)/APS Outputs/PhiE 0Y2 <-> Data Pointer/PhiSetPoints[5]
//     Term 23 (APS4322-7000)/APS Outputs/PhiE 1Y0 <-> Data Pointer/PhiSetPoints[9]
//     Term 23 (APS4322-7000)/APS Outputs/PhiE 1Y1 <-> Data Pointer/PhiSetPoints[10]
//     Term 23 (APS4322-7000)/APS Outputs/PhiE 1Y2 <-> Data Pointer/PhiSetPoints[11]
//     Term 23 (APS4322-7000)/APS Outputs/PhiE 2Y0 <-> Data Pointer/PhiSetPoints[15]
//     Term 23 (APS4322-7000)/APS Outputs/PhiE 2Y1 <-> Data Pointer/PhiSetPoints[16]
//     Term 23 (APS4322-7000)/APS Outputs/PhiE 2Y2 <-> Data Pointer/PhiSetPoints[17]
//     Term 23 (APS4322-7000)/APS Outputs/PhiE 3Y0 <-> Data Pointer/PhiSetPoints[21]
//     Term 23 (APS4322-7000)/APS Outputs/PhiE 3Y1 <-> Data Pointer/PhiSetPoints[22]
//     Term 23 (APS4322-7000)/APS Outputs/PhiE 3Y2 <-> Data Pointer/PhiSetPoints[23]
//     Term 23 (APS4322-7000)/Term 24 (APS4322-5000)/FB Inputs/A{0..8 step 2} X-Field <-> Data Pointer/HallSensorFieldsXYZ[{0..12 step 3}]  (5 links)
//     Term 23 (APS4322-7000)/Term 24 (APS4322-5000)/FB Inputs/A{0..8 step 2} Y-Field <-> Data Pointer/HallSensorFieldsXYZ[{1..13 step 3}]  (5 links)
//     Term 23 (APS4322-7000)/Term 24 (APS4322-5000)/FB Inputs/A{0..8 step 2} Z-Field <-> Data Pointer/HallSensorFieldsXYZ[{2..14 step 3}]  (5 links)
//     Term 23 (APS4322-7000)/Term 24 (APS4322-5000)/FB Inputs/B{1..9 step 2} X-Field <-> Data Pointer/HallSensorFieldsXYZ[{15..27 step 3}]  (5 links)
//     Term 23 (APS4322-7000)/Term 24 (APS4322-5000)/FB Inputs/B{1..9 step 2} Y-Field <-> Data Pointer/HallSensorFieldsXYZ[{16..28 step 3}]  (5 links)
//     Term 23 (APS4322-7000)/Term 24 (APS4322-5000)/FB Inputs/B{1..9 step 2} Z-Field <-> Data Pointer/HallSensorFieldsXYZ[{17..29 step 3}]  (5 links)
//     Term 23 (APS4322-7000)/Term 24 (APS4322-5000)/FB Inputs/C{0..8 step 2} X-Field <-> Data Pointer/HallSensorFieldsXYZ[{30..42 step 3}]  (5 links)
//     Term 23 (APS4322-7000)/Term 24 (APS4322-5000)/FB Inputs/C{0..8 step 2} Y-Field <-> Data Pointer/HallSensorFieldsXYZ[{31..43 step 3}]  (5 links)
//     Term 23 (APS4322-7000)/Term 24 (APS4322-5000)/FB Inputs/C{0..8 step 2} Z-Field <-> Data Pointer/HallSensorFieldsXYZ[{32..44 step 3}]  (5 links)
//     Term 23 (APS4322-7000)/Term 24 (APS4322-5000)/FB Inputs/D{1..9 step 2} X-Field <-> Data Pointer/HallSensorFieldsXYZ[{45..57 step 3}]  (5 links)
//     Term 23 (APS4322-7000)/Term 24 (APS4322-5000)/FB Inputs/D{1..9 step 2} Y-Field <-> Data Pointer/HallSensorFieldsXYZ[{46..58 step 3}]  (5 links)
//     Term 23 (APS4322-7000)/Term 24 (APS4322-5000)/FB Inputs/D{1..9 step 2} Z-Field <-> Data Pointer/HallSensorFieldsXYZ[{47..59 step 3}]  (5 links)
//     Term 23 (APS4322-7000)/Term 24 (APS4322-5000)/FB Inputs/E{0..8 step 2} X-Field <-> Data Pointer/HallSensorFieldsXYZ[{60..72 step 3}]  (5 links)
//     Term 23 (APS4322-7000)/Term 24 (APS4322-5000)/FB Inputs/E{0..8 step 2} Y-Field <-> Data Pointer/HallSensorFieldsXYZ[{61..73 step 3}]  (5 links)
//     Term 23 (APS4322-7000)/Term 24 (APS4322-5000)/FB Inputs/E{0..8 step 2} Z-Field <-> Data Pointer/HallSensorFieldsXYZ[{62..74 step 3}]  (5 links)
//     Term 23 (APS4322-7000)/Term 24 (APS4322-5000)/FB Inputs/F{1..9 step 2} X-Field <-> Data Pointer/HallSensorFieldsXYZ[{75..87 step 3}]  (5 links)
//     Term 23 (APS4322-7000)/Term 24 (APS4322-5000)/FB Inputs/F{1..9 step 2} Y-Field <-> Data Pointer/HallSensorFieldsXYZ[{76..88 step 3}]  (5 links)
//     Term 23 (APS4322-7000)/Term 24 (APS4322-5000)/FB Inputs/F{1..9 step 2} Z-Field <-> Data Pointer/HallSensorFieldsXYZ[{77..89 step 3}]  (5 links)
//     Term 23 (APS4322-7000)/Term 24 (APS4322-5000)/FB Inputs/G{0..8 step 2} X-Field <-> Data Pointer/HallSensorFieldsXYZ[{90..102 step 3}]  (5 links)
//     Term 23 (APS4322-7000)/Term 24 (APS4322-5000)/FB Inputs/G{0..8 step 2} Y-Field <-> Data Pointer/HallSensorFieldsXYZ[{91..103 step 3}]  (5 links)
//     Term 23 (APS4322-7000)/Term 24 (APS4322-5000)/FB Inputs/G{0..8 step 2} Z-Field <-> Data Pointer/HallSensorFieldsXYZ[{92..104 step 3}]  (5 links)
//     Term 23 (APS4322-7000)/Term 24 (APS4322-5000)/FB Inputs/H{1..9 step 2} X-Field <-> Data Pointer/HallSensorFieldsXYZ[{105..117 step 3}]  (5 links)
//     Term 23 (APS4322-7000)/Term 24 (APS4322-5000)/FB Inputs/H{1..9 step 2} Y-Field <-> Data Pointer/HallSensorFieldsXYZ[{106..118 step 3}]  (5 links)
//     Term 23 (APS4322-7000)/Term 24 (APS4322-5000)/FB Inputs/H{1..9 step 2} Z-Field <-> Data Pointer/HallSensorFieldsXYZ[{107..119 step 3}]  (5 links)
//     Term 23 (APS4322-7000)/Term 24 (APS4322-5000)/FB Inputs/I{0..8 step 2} X-Field <-> Data Pointer/HallSensorFieldsXYZ[{120..132 step 3}]  (5 links)
//     Term 23 (APS4322-7000)/Term 24 (APS4322-5000)/FB Inputs/I{0..8 step 2} Y-Field <-> Data Pointer/HallSensorFieldsXYZ[{121..133 step 3}]  (5 links)
//     Term 23 (APS4322-7000)/Term 24 (APS4322-5000)/FB Inputs/I{0..8 step 2} Z-Field <-> Data Pointer/HallSensorFieldsXYZ[{122..134 step 3}]  (5 links)
//     Term 23 (APS4322-7000)/Term 24 (APS4322-5000)/FB Inputs/J{1..9 step 2} X-Field <-> Data Pointer/HallSensorFieldsXYZ[{135..147 step 3}]  (5 links)
//     Term 23 (APS4322-7000)/Term 24 (APS4322-5000)/FB Inputs/J{1..9 step 2} Y-Field <-> Data Pointer/HallSensorFieldsXYZ[{136..148 step 3}]  (5 links)
//     Term 23 (APS4322-7000)/Term 24 (APS4322-5000)/FB Inputs/J{1..9 step 2} Z-Field <-> Data Pointer/HallSensorFieldsXYZ[{137..149 step 3}]  (5 links)
//     Term 23 (APS4322-7000)/Term 24 (APS4322-5000)/FB Inputs/Status <-> Data Pointer/FeedbackStatus
//   XPlanar MC Project/Axes/Mover4330_1 <-> TcCOM Objects/XPlanar/Mover4330_1
//     IoToMc/STD <-> OutputsToNC3/HWToNC3
//   XPlanar MC Project/Axes/Mover4330_2 <-> TcCOM Objects/XPlanar/Mover4330_2
//     McToIo/STD <-> InputsFromNC3/NC3ToHW
//   XPlanar MC Project/Axes/Mover4330_3 <-> TcCOM Objects/XPlanar/Mover4330_3
//     IoToMc/STD <-> OutputsToNC3/HWToNC3
//     McToIo/STD <-> InputsFromNC3/NC3ToHW
//   XPlanar MC Project/Axes/Mover4330_4 <-> TcCOM Objects/XPlanar/Mover4330_4
//     McToIo/STD <-> InputsFromNC3/NC3ToHW
//   SMXPlanarMoverTest/SMXPlanarMoverTest Instance <-> Device 1 (EtherCAT)/Term 1 (EK1200)/Term 2 (EL9222-9482)
//     PlcTask Inputs/MAIN.EL9222_9482.MDP5001_922_Input/MDP5001_922_OCP_Inputs_Channel_1_Status <-> OCP Inputs Channel 2/Status
//   SMXPlanarMoverTest/SMXPlanarMoverTest Instance <-> Device 1 (EtherCAT)/Term 1 (EK1200)/Term 3 (EL9222-6600)
//     PlcTask Inputs/MAIN.EL9222_6600.MDP5001_922_Input/MDP5001_922_OCP_Inputs_Channel_1_Status <-> OCP Inputs Channel 2/Status
//   SMXPlanarMoverTest/SMXPlanarMoverTest Instance <-> XPlanar MC Project/Axes/Mover4330_1
//     PlcTask Inputs/MAIN.fbMover1.MCTOPLC/ACT <-> McToPlc/ACT
//     PlcTask Inputs/MAIN.fbMover1.MCTOPLC/COORDMODE <-> McToPlc/COORDMODE
//     PlcTask Inputs/MAIN.fbMover1.MCTOPLC/SET <-> McToPlc/SET
//     PlcTask Inputs/MAIN.fbMover1.MCTOPLC/SETONTRACK <-> McToPlc/SETONTRACK
//     PlcTask Inputs/MAIN.fbMover1.MCTOPLC/STD <-> McToPlc/STD
//     PlcTask Outputs/MAIN.fbMover1.PLCTOMC/STD <-> PlcToMc/STD
//   SMXPlanarMoverTest/SMXPlanarMoverTest Instance <-> XPlanar MC Project/Axes/Mover4330_2
//     PlcTask Inputs/MAIN.fbMover2.stMoverRef.MCTOPLC/ACT <-> McToPlc/ACT
//     PlcTask Inputs/MAIN.fbMover2.stMoverRef.MCTOPLC/COORDMODE <-> McToPlc/COORDMODE
//     PlcTask Inputs/MAIN.fbMover2.stMoverRef.MCTOPLC/SET <-> McToPlc/SET
//     PlcTask Inputs/MAIN.fbMover2.stMoverRef.MCTOPLC/SETONTRACK <-> McToPlc/SETONTRACK
//     PlcTask Inputs/MAIN.fbMover2.stMoverRef.MCTOPLC/STD <-> McToPlc/STD
//     PlcTask Outputs/MAIN.fbMover2.stMoverRef.PLCTOMC/STD <-> PlcToMc/STD
//   SMXPlanarMoverTest/SMXPlanarMoverTest Instance <-> XPlanar MC Project/Axes/Mover4330_3
//     PlcTask Inputs/MAIN.fbMover3.stMoverRef.MCTOPLC/ACT <-> McToPlc/ACT
//     PlcTask Inputs/MAIN.fbMover3.stMoverRef.MCTOPLC/COORDMODE <-> McToPlc/COORDMODE
//     PlcTask Inputs/MAIN.fbMover3.stMoverRef.MCTOPLC/SET <-> McToPlc/SET
//     PlcTask Inputs/MAIN.fbMover3.stMoverRef.MCTOPLC/SETONTRACK <-> McToPlc/SETONTRACK
//     PlcTask Inputs/MAIN.fbMover3.stMoverRef.MCTOPLC/STD <-> McToPlc/STD
//     PlcTask Outputs/MAIN.fbMover3.stMoverRef.PLCTOMC/STD <-> PlcToMc/STD
//   SMXPlanarMoverTest/SMXPlanarMoverTest Instance <-> XPlanar MC Project/Axes/Mover4330_4
//     PlcTask Inputs/MAIN.fbMover4.stMoverRef.MCTOPLC/ACT <-> McToPlc/ACT
//     PlcTask Inputs/MAIN.fbMover4.stMoverRef.MCTOPLC/COORDMODE <-> McToPlc/COORDMODE
//     PlcTask Inputs/MAIN.fbMover4.stMoverRef.MCTOPLC/SET <-> McToPlc/SET
//     PlcTask Inputs/MAIN.fbMover4.stMoverRef.MCTOPLC/SETONTRACK <-> McToPlc/SETONTRACK
//     PlcTask Inputs/MAIN.fbMover4.stMoverRef.MCTOPLC/STD <-> McToPlc/STD
//     PlcTask Outputs/MAIN.fbMover4.stMoverRef.PLCTOMC/STD <-> PlcToMc/STD
//   SMXPlanarMoverTest/SMXPlanarMoverTest Instance <-> XPlanar MC Project/Groups/Environment
//     PlcTask Inputs/MAIN.fbEnvironment.MCTOPLC_STD <-> McToPlc/STD
//   SMXPlanarMoverTest/SMXPlanarMoverTest Instance <-> XPlanar MC Project/Groups/XPlanar
//     PlcTask Inputs/MAIN.fbGroup.MCTOPLC_STD <-> McToPlc/STD
//   StarterkitApplicationPLC/StarterkitApplicationPLC Instance <-> Device 1 (EtherCAT)/Term 1 (EK1200)/Term 2 (EL9222-9482)
//     PlcTask Inputs/MAIN.stEL9222_1_Status <-> OCP Inputs Channel 1/Status
//   StarterkitApplicationPLC/StarterkitApplicationPLC Instance <-> Device 1 (EtherCAT)/Term 1 (EK1200)/Term 3 (EL9222-6600)
//     PlcTask Inputs/MAIN.stEL9222_2_Status <-> OCP Inputs Channel 1/Status
//   TcCOM Objects/XPlanar/Mover4330_1 <-> XPlanar MC Project/Axes/Mover4330_1
//     InputsFromNC3/NC3ToHW <-> McToIo/STD
//   TcCOM Objects/XPlanar/Mover4330_2 <-> XPlanar MC Project/Axes/Mover4330_2
//     OutputsToNC3/HWToNC3 <-> IoToMc/STD
//   TcCOM Objects/XPlanar/Mover4330_4 <-> XPlanar MC Project/Axes/Mover4330_4
//     OutputsToNC3/HWToNC3 <-> IoToMc/STD

CONFIGURATION StarterkitApplicationPLC
    RESOURCE PLC ON TwinCAT3
        TASK PlcTask(INTERVAL := T#2ms, PRIORITY := 20);
        PROGRAM MAIN WITH PlcTask : MAIN;
    END_RESOURCE
END_CONFIGURATION

// ---- 1_Industry/DUTs/E_XMotion_Command.TcDUT
{attribute 'qualified_only'}
{attribute 'strict'}
TYPE E_XMotion_Command :
(
	NoCommand		:= 0,
	Abort			:= 1,
	Reset			:= 2,
	Prepare			:= 3,
	Start			:= 4,
	HoldOnError		:= 5,
	UserCommand		:= 6
	
) DINT;
END_TYPE

// ---- 1_Industry/DUTs/E_XMotion_Status.TcDUT
{attribute 'qualified_only'}
{attribute 'strict'}
TYPE E_XMotion_Status :
(
	StartUp 	:= 0,
	Aborting 	:= 1,
	Aborted 	:= 2,	
	Resetting   := 3,
	Stopped  	:= 4,
	Preparing   := 5,
	Prepared    := 6,
	Execute 	:= 7,
	HoldOnError := 8
	
) DINT;
END_TYPE

// ---- 1_Industry/DUTs/ST_VisControl.TcDUT
TYPE ST_VisControl :
STRUCT
	
	stControlPad	: ST_Vis_ControlPadControl;
	stOperatorPad	: ST_Vis_OperationalControl;


END_STRUCT
END_TYPE

// ---- 1_Industry/DUTs/ST_Vis_ControlPadControl.TcDUT
TYPE ST_Vis_ControlPadControl :
STRUCT
	
	bVisInvisibleButton	: BOOL;	
	bVisInvisible		: BOOL;	
	nFramePositionX		: INT;
	nFramePositionY		: INT;
	nButtonPositionX	: INT;
	nButtonPositionY	: INT;
	
	bButtonState_Abort			: BOOL;
	bButtonState_Reset			: BOOL;
	bButtonState_Prepare		: BOOL;	
	bButtonState_Start			: BOOL;
	
	bStateSignalAbortBlue		: BOOL;
	bStateSignalAbortYellow		: BOOL;
	bStateSignalAbortGreen		: BOOL;
	
	bStateSignalResetYellow		: BOOL;
	bStateSignalResetGreen		: BOOL;

	bStateSignalPrepareYellow	: BOOL;
	bStateSignalPrepareGreen	: BOOL;

	bStateSignalExecuteYellow	: BOOL;
	bStateSignalExecuteGreen	: BOOL;	

	bAbortSequenceStateInvisible	: BOOL;
	bResetSequenceStateInvisible	: BOOL;
	bPrepareSequenceStateInvisible	: BOOL;
	bStartSequenceStateInvisible	: BOOL;
	
	iAbortSequenceState			: INT;
	iResetSequenceState			: INT;
	iPrepareSequenceState		: INT;
	iStartSequenceState			: INT;	
	
	
END_STRUCT
END_TYPE

// ---- 1_Industry/DUTs/ST_Vis_OperationalControl.TcDUT
TYPE ST_Vis_OperationalControl :
STRUCT
	bVisInvisibleButton	: BOOL;	
	bVisInvisible		: BOOL;
	nFramePositionX		: REAL;
	nFramePositionY		: REAL;
	nButtonPositionX	: INT;
	nButtonPositionY	: INT;	
	
	bStartButtunState	: BOOL;
	bStopButtonState	: BOOL;
	bQuitButtonState	: BOOL;
	bEStopButtonState	: BOOL;
	
	bStartButtonLamp	: BOOL;
	bStopButtonLamp		: BOOL;
	bQuitButtonLamp		: BOOL;
	bEStopButtonLamp	: BOOL;
	
	bMessageColorGreen	: BOOL;
	bMessageColorRed	: BOOL;
	
	sMessage			: STRING;
	
	
END_STRUCT
END_TYPE

// ---- 1_Industry/DUTs/ST_XMotionStatemachineStates.TcDUT
TYPE ST_XMotionStatemachineStates :
STRUCT
	nAbortState		: INT;
	nResetState		: INT;
	nPrepareState	: INT;
	nStartState		: INT;
END_STRUCT
END_TYPE

// ---- 1_Industry/DUTs/ST_XTags.TcDUT
TYPE ST_XTags :
STRUCT
	

	Command		: E_XMotion_Command;
	Status		: E_XMotion_Status;
	States		: ST_XMotionStatemachineStates;
	
END_STRUCT
END_TYPE

// ---- 2_Application/Machine/DUTs/ST_MachineState.TcDUT
TYPE ST_MachineState :
STRUCT

	bStartup	 : BOOL;		
	bStartupDone : BOOL;
	bAborting 	 : BOOL;
	bResetting	 : BOOL;
	bStarting	 : BOOL;
	bRunning	 : BOOL;

END_STRUCT
END_TYPE

// ---- 2_Application/Mover/DUTs/ST_ProductData.TcDUT
TYPE ST_ProductData :
STRUCT
	
	nSerial				: UDINT;
	bInitRun			: BOOL;
	nDestinationProcess	: UINT;
	nPriority			: UINT;
	

END_STRUCT
END_TYPE

// ---- 2_Application/Station/DUTs/ST_StationReturn.TcDUT
TYPE ST_StationReturn :
STRUCT
	Done	: BOOL;
	stState	: INT;
END_STRUCT
END_TYPE

// ---- 2_Application/Station/DUTs/ST_StationTrackPosition.TcDUT
TYPE ST_StationTrackPosition :
STRUCT
	fPositionOnTrack	: LREAL;
	nTrackId			: INT;	
END_STRUCT
END_TYPE

// ---- 1_Industry/GlobalVariables.TcGVL


VAR_GLOBAL
	
	XTags			: ST_XTags;		

	stVisControl	: ST_VisControl;
	

END_VAR

// ---- 2_Application/GVL_Application.TcGVL
VAR_GLOBAL CONSTANT
	
	MaxMovers			: UDINT := 4;		// Number of movers to control
	trackCount			: UDINT := 3;		// Number of tracks controlled by the application
	nStationCount		: UINT  := 5;		// Number of stations controlled by the application
	maxNumTrackPoints	: INT   := 20;		// max number of track points for each track 
END_VAR

VAR_GLOBAL
	moverCount					: UDINT := 4;
	ipTrack						: ARRAY [1..trackCount] OF I_Track;
	ipStation					: ARRAY [1..nStationCount] OF I_Station;
	ipMoverApplication			: ARRAY [1..MaxMovers] OF I_MoverApplication;
	ipMotionSystemApplication	: I_MotionSystemApplication;
	ipXpu						: I_TcIoXPlanarProcessingUnit;
END_VAR

// ---- 2_Application/Machine/I_MotionSystemApplication.TcIO
INTERFACE I_MotionSystemApplication

METHOD Aborting : BOOL
VAR_INPUT
END_VAR
END_METHOD

METHOD Cycle : BOOL
VAR_INPUT
END_VAR
END_METHOD

METHOD Execute : UDINT
VAR_INPUT
END_VAR
END_METHOD

PROPERTY P_bMoverError : BOOL
GET
END_GET
SET
END_SET
END_PROPERTY

PROPERTY PUBLIC P_nAbortingSequence : UDINT
GET
END_GET
END_PROPERTY

PROPERTY PUBLIC P_nExecutingSequence : UDINT
GET
END_GET
END_PROPERTY

PROPERTY PUBLIC P_nResettingSequence : UDINT
GET
END_GET
END_PROPERTY

PROPERTY PUBLIC P_nStartingSequence : UDINT
GET
END_GET
END_PROPERTY

PROPERTY PUBLIC P_nStartupSequence : UDINT
GET
END_GET
END_PROPERTY

METHOD Resetting : BOOL
VAR_INPUT
END_VAR
END_METHOD

METHOD Starting : BOOL
VAR_INPUT
END_VAR
END_METHOD

METHOD Startup : BOOL
VAR_INPUT
END_VAR
END_METHOD

PROPERTY std : I_MotionSystem
GET
END_GET
SET
END_SET
END_PROPERTY

END_INTERFACE

// ---- 2_Application/Mover/I_MoverApplication.TcIO
INTERFACE I_MoverApplication

METHOD Cycle
END_METHOD

PROPERTY P_nMoverIndex : INT
GET
END_GET
SET
END_SET
END_PROPERTY

PROPERTY P_nTrackId : UDINT
GET
END_GET
SET
END_SET
END_PROPERTY

PROPERTY ProductData : Reference to ST_ProductData
GET
END_GET
SET
END_SET
END_PROPERTY

PROPERTY std : I_XPlanarMoverStandard
GET
END_GET
SET
END_SET
END_PROPERTY

END_INTERFACE

// ---- 2_Application/Station/I_Station.TcIO
INTERFACE I_Station

METHOD ccl00_cycle : BOOL
VAR_INPUT
END_VAR
END_METHOD

METHOD ClearList : BOOL
VAR_INPUT
END_VAR
END_METHOD

PROPERTY InputConnections : I_Station
GET
END_GET
SET
END_SET
END_PROPERTY

PROPERTY OutputConnections : I_Station
GET
END_GET
SET
END_SET
END_PROPERTY

PROPERTY P_List : I_List
GET
END_GET
END_PROPERTY

PROPERTY P_List_Input_B : I_List
GET
END_GET
END_PROPERTY

PROPERTY P_List_Input_C : I_List
GET
END_GET
END_PROPERTY

PROPERTY P_nErrorCode : UDINT
GET
END_GET
END_PROPERTY

PROPERTY P_PositionOnTrack : ST_StationTrackPosition
GET
END_GET
END_PROPERTY

METHOD Processing : BOOL
VAR_INPUT
	i_nMachineState 	: INT;		// 1=Starting, 2=Running
END_VAR
END_METHOD

METHOD ResetStation : BOOL
VAR_INPUT
	bClear	: BOOL;
END_VAR
END_METHOD

END_INTERFACE

// ---- 2_Application/Tracks/I_Track.TcIO
INTERFACE I_Track

METHOD ccl00_cycle : BOOL
END_METHOD

METHOD Initialize : BOOL
VAR_INPUT
	bExecute 			: BOOL;
END_VAR
END_METHOD

PROPERTY P_TrackLength : LREAL
GET
END_GET
END_PROPERTY

PROPERTY std : I_TrackStandard
GET
END_GET
END_PROPERTY

END_INTERFACE

// ---- MAIN.TcPOU
{attribute 'TcCallAfterOutputUpdate'}
PROGRAM MAIN

VAR
// MAIN
	fbXMotionUnit					: FB_MachineModule;
	fbOperationalControl			: FB_OperationalControl;
	fbVisStarterKitStateMachine		: FB_VisStarterKitStateMachine;	
	
	bExternalMachineStop : BOOL;
	
	bHelp01		: BOOL;
	bHelp02		: BOOL;	
	bHelp03		: BOOL;
	bHelp04		: BOOL;	
	sHelp01		: STRING;
	nHelp01		: INT;
	
	
	
	dcTimeStamp AT%Q*		: ULINT;
	

	// Track Plotter
	nTestCnt				: UINT;
	bTrackPlot				: BOOL;
	nForCounter				: INT;
	position				: PositionXYC;
	fTrackPointDistance1 	: LREAL;
	fTrackPointDistance2	: LREAL;
	fTrackPointDistance3	: LREAL;
	fTrackPointDistance4	: LREAL;
	
	arTrackPoints1 		: ARRAY [1..1000,1..2] OF LREAL;
	arTrackPoints2 		: ARRAY [1..1000,1..2] OF LREAL;
	arTrackPoints3 		: ARRAY [1..1000,1..2] OF LREAL;
	arTrackPoints4 		: ARRAY [1..1000,1..2] OF LREAL;

	stEL9222_1_Status	AT %I*	: DWORD;
	stEL9222_2_Status	AT %I*	: DWORD;
	
END_VAR

Cycle();

METHOD Cycle : BOOL
VAR_INPUT
END_VAR
fbXMotionUnit.Cycle(); 									// Keep it alive!            

fbXMotionUnit.XCommand := XTags.Command;	    		// Writing command from superior unit e.g. HMI
XTags.Status := fbXMotionUnit.XMotionStatus;			// Getting current status of XMotionUnit for e.g. HMI display	
XTags.States := fbXMotionUnit.XSequenceStates; 			// Writing current states information into XTags
fbXMotionUnit.bExternelStop := bExternalMachineStop;	// External exception e.g. signal from E-Stop


fbXMotionUnit.P_bErrorQuit := fbVisStarterKitStateMachine.bOCQuitButtonState;
fbOperationalControl.P_nProcessFeedback := fbXMotionUnit.P_nProcessFeedback;


fbOperationalControl(	   bStartCommand := fbVisStarterKitStateMachine.bOCStartButtonState, 
					        bStopCommand := fbVisStarterKitStateMachine.bOCStopButtonState, 
						    bQuitCommand := fbVisStarterKitStateMachine.bOCQuitButtonState,
					   bExceptionCommand := fbVisStarterKitStateMachine.bOCEStopButtonState,
							  bStartLamp => bHelp01,
							   bStopLamp => bHelp02,
                               bQuitLamp => bHelp03,
                              bEStopLamp => bHelp04,
							    bStopped => ,
							   bStarting => , 
							    bRunning => , 
							     sResult => sHelp01,
							     nResult => nHelp01,
							       XTags := XTags );
	

							fbVisStarterKitStateMachine.bOCStartLampState 		:= bHelp01;
							fbVisStarterKitStateMachine.bOCStopLampState  		:= bHelp02;
							fbVisStarterKitStateMachine.bOCQuitLampState  		:= bHelp03;
							fbVisStarterKitStateMachine.bOCEStopLampState  	 	:= bHelp04;
							fbVisStarterKitStateMachine.sOCResultTextDisplay 	:= sHelp01;
							fbVisStarterKitStateMachine.nOCResult 				:= nHelp01;							  
									  
	fbVisStarterKitStateMachine( iq_stVisControl := stVisControl,
                         				iq_XTags := XTags );
END_METHOD

END_PROGRAM

// ---- 1_Industry/FB_MachineModule.TcPOU

//The functionblock FB_Generick is transmitted to every Machine-Unit

FUNCTION_BLOCK FB_MachineModule 

VAR
//===== application layer =================================

	fbMotionSystem			: FB_MotionSystem;
 	{IF defined (XPlanar)}
	fbXPlanarSystem			: FB_XPlanarSystem;
	{ELSIF defined (XTS)}
	fbXtsSystem				: FB_XtsSystem;
	{END_IF}

	fbMover					: ARRAY [1..MaxMovers] OF FB_ApplicationMover;
	{IF defined (XPlanar)}
	fbXPlanarMover			: ARRAY [1..MaxMovers] OF FB_XPlanarMoverStandard; 
	{ELSIF defined (XTS)}	
	fbXtsMover				: ARRAY [1..moverCount] OF FB_XtsMover; 	
	{END_IF}

	// Instances of Track-FBs
	fbTrackSegment01		: FB_TrackSegment_1;
	fbTrackSegment02		: FB_TrackSegment_2;
	fbTrackSegment03		: FB_TrackSegment_3;
	   
	// Instances of Station-FBs
	fbStation_01_Process 	: FB_Station_01_Process;
	fbStation_02_Process 	: FB_Station_02_Process;
	fbStation_03_Process	: FB_Station_03_Process;
	fbStation_04_Switch		: FB_Station_04_SW_Separate;
	fbStation_05_Switch		: FB_Station_05_SW_Merge;
	
	
//=========================================================

	tonPowerOnDelayOff		: TON;
	bPowerOnDelayOff		: BOOL;
	ObPowerOn	AT%Q* : BOOL := FALSE;

//===== base module =======================================
	eXCommand					: E_XMotion_Command;
	eXStatus					: E_XMotion_Status;
	eLastXState					: E_XMotion_Status;	

	
	fbStateManager				: FB_SK_StateManager;
	eControlCommand				: E_XMotion_Command;
	stSequenceStates 			: ST_XMotionStatemachineStates;
	
	nStateCommandCheck			: INT;
	bMachineExceptionPending	: BOOL;
	
	bUnitModeManagerExecute		: BOOL;
	bUnitModeManagerDone		: BOOL;
	bUnitModeManagerError		: BOOL;
	
	DelayTimerDemo				: TON;
	
	nStateSequence				: INT;
	nStateExecute				: INT;
	bInterfaceAssignmentDone	: BOOL;
	bDone						: BOOL;
	
	nProcessFeedback			: UDINT;
	bErrorQuit					: BOOL;
	
	nForCounter					: UDINT;

	
	// ...just for testing 
	nTestCounter_Cycle				: UINT;
	nTestCounter_Aborted			: UINT;
	nTestCounter_Aborting			: UINT;
	nTestCounter_Execute			: UINT;
	nTestCounter_Preparing			: UINT;
	nTestCounter_Prepared			: UINT;
	nTestCounter_Resetting 			: UINT;
	nTestCounter_StartUp			: UINT;
	nTestCounter_StateComplete 		: UINT;
	nTestCounter_Stopped			: UINT;
	nTestCounter_CommandReceive		: UINT;	
	
	fbVisu : FB_XPlanarVisuDiag;
	
	binit : BOOL;
	
END_VAR

{attribute 'object_name' := 'Aborted'}
METHOD PRIVATE Aborted



	nTestCounter_Aborted := nTestCounter_Aborted + 1;
	
	(*
		Aborted:
		- all movers deactivated
		- No errors pending
	*)
END_METHOD

{attribute 'object_name' := 'Aborting'}
METHOD PRIVATE Aborting
CASE nStateSequence OF
	0: 		
		IF ipMotionSystemApplication <> 0 THEN
			nStateSequence := 10;
		END_IF


	10:	
		bDone := ipMotionSystemApplication.Aborting();

		IF bDone THEN
			nStateSequence := 100;
		END_IF

	100:
		StateComplete();
END_CASE
END_METHOD

PROPERTY bExternelStop : BOOL
GET
END_GET
SET
END_SET
END_PROPERTY

METHOD PRIVATE CommandReceive 
VAR_INPUT
END_VAR


	nTestCounter_CommandReceive := nTestCounter_CommandReceive + 1;


	
	// Checking Statecommands and reacting to received Control-Commands
	CASE nStateCommandCheck OF
	
	
	0:  // Check
		IF NOT bMachineExceptionPending THEN
			nStateCommandCheck:= 10;   	// No error
		ELSE
			nStateCommandCheck:= 20;	// Error pending
		END_IF
	
		
	10:	// No Machine-Error 
		
		CASE eXCommand OF 		// XTags.eCommand received from superior system e.g. Machine-HMI

		E_XMotion_Command.NoCommand:
				eControlCommand := E_XMotion_Command.NoCommand;
		
		E_XMotion_Command.Abort:
				eControlCommand := E_XMotion_Command.Abort;
		
		E_XMotion_Command.Reset: 
				IF eXStatus = E_XMotion_Status.Aborted THEN
					eControlCommand := E_XMotion_Command.Reset;
				END_IF		
		
		E_XMotion_Command.Prepare:
				IF eXStatus = E_XMotion_Status.Stopped THEN
					eControlCommand := E_XMotion_Command.Prepare;
				END_IF
	
		E_XMotion_Command.Start:	
				IF eXStatus = E_XMotion_Status.Prepared THEN
					eControlCommand := E_XMotion_Command.Start;
				END_IF		
			
		E_XMotion_Command.HoldOnError:
				eControlCommand := E_XMotion_Command.HoldOnError;

				
		E_XMotion_Command.UserCommand:
				;
		
		// Rückmeldung wenn/warum ein Command nicht ausgeführt wurde		
							
		END_CASE
				
		nStateCommandCheck := 0;	
	
		
	20:  // Machine-Error reaction
		   eControlCommand := E_XMotion_Command.Abort;
		nStateCommandCheck := nStateCommandCheck + 1;	
		
	21: IF XTags.Status = E_XMotion_Status.Aborted THEN
			nStateCommandCheck := nStateCommandCheck + 1;
		END_IF		
			
	22:	IF NOT bMachineExceptionPending THEN
			nStateCommandCheck := 10;
		END_IF
		
		
	END_CASE
END_METHOD

METHOD PUBLIC Cycle
VAR
	nForCounter : UDINT;	
END_VAR
	{IF defined (XPlanar)}	
	fbMotionSystem.std := THIS^.fbXPlanarSystem;
	{ELSIF defined (XTS)}
	fbMotionSystem.std := THIS^.fbXtsSystem;
	{END_IF}


	// Checking for command received by superior unit e.g. HMI
	CommandReceive();
		
	// fbStateManager manages the state to be executed:
	fbStateManager.Cycle();	
	fbStateManager.XMotionCommand := eControlCommand;
	eXStatus := fbStateManager.Status;
						
	IF eXStatus <> eLastXState THEN
		nStateSequence := 0;
		eLastXState := eXStatus;
	END_IF

	// One of the methods is executing by the actual status
	CASE eXStatus OF
		E_XMotion_Status.StartUp:	        StartUp();
		E_XMotion_Status.Aborting:         Aborting();
		E_XMotion_Status.Aborted:           Aborted();
		E_XMotion_Status.Resetting:       Resetting();
		E_XMotion_Status.Stopped:           Stopped();
		E_XMotion_Status.Preparing:       Preparing();
		E_XMotion_Status.Prepared:         Prepared();
		E_XMotion_Status.Execute:	   		Execute();
		E_XMotion_Status.HoldOnError:	HoldOnError();
	END_CASE

	// E-Stop PowerOff
	tonPowerOnDelayOff(IN:=eXStatus=E_XMotion_Status.Aborting OR eXStatus=E_XMotion_Status.Aborted OR eXStatus=E_XMotion_Status.StartUp , PT:=T#5H , Q=> , ET=> );
	bPowerOnDelayOff := NOT tonPowerOnDelayOff.Q;
	ObPowerOn := bPowerOnDelayOff;
	
	// Information to visulization etc.
	IF ipMotionSystemApplication <> 0 THEN 
		stSequenceStates.nAbortState   := UDINT_TO_INT(ipMotionSystemApplication.P_nAbortingSequence); 
		stSequenceStates.nResetState   := UDINT_TO_INT(ipMotionSystemApplication.P_nResettingSequence);
		stSequenceStates.nPrepareState := UDINT_TO_INT(ipMotionSystemApplication.P_nStartingSequence);
		stSequenceStates.nStartState   := UDINT_TO_INT(ipMotionSystemApplication.P_nExecutingSequence);
	END_IF	
	
	
	
	// Keeping all cyclic activities alive
	IF ipMotionSystemApplication <> 0 THEN
		ipMotionSystemApplication.std.Cycle();
		ipMotionSystemApplication.Cycle();
	END_IF
	
	FOR nForCounter := 1 TO moverCount DO
		IF ipMoverApplication[nforcounter] <> 0 THEN
			ipMotionSystemApplication.std.SetMoverStandard(nforcounter,ipMoverApplication[nForCounter].std);
			ipMoverApplication[nForCounter].std.P_Id :=UDINT_TO_UINT(nForCounter);
			ipMoverApplication[nforcounter].Cycle();
		END_IF
	END_FOR		
	
	FOR nForCounter:=1 TO nStationCount DO 
		IF ipStation[nForCounter] <> 0 THEN 
			ipStation[nForCounter].ccl00_cycle(); 
		END_IF
	END_FOR	
	
	FOR nForCounter := 1 TO trackCount DO
		IF ipTrack[nForCounter] <> 0 THEN
			ipMotionSystemApplication.std.SetTrackStandard(nForCounter, ipTrack[nForCounter].std);
			ipTrack[nForCounter].ccl00_cycle();
		END_IF
	END_FOR



//Visu
IF NOT bInit THEN
	IF ipMoverApplication[1] <> 0 THEN
		binit := TRUE;
		FOR nForCounter := 1 TO 4 DO 
			IF ipMoverApplication[nForCounter] <> 0 THEN
				fbVisu.SetStandardMover(ipMoverApplication[nForCounter].std, UDINT_TO_INT(nForCounter));
			END_IF
		END_FOR
	END_IF
END_IF
fbVisu.UpdateMoverStatus();
END_METHOD

{attribute 'object_name' := 'Execute'}
METHOD PRIVATE Execute


	
VAR_INST
	nForCounter : UDINT;	


END_VAR

	
	FOR nForCounter:=1 TO nStationCount DO
		IF ipStation[nForCounter] <> 0 THEN
			ipStation[nForCounter].Processing(i_nMachineState:=2);
			
			IF ipStation[nForCounter].P_nErrorCode > 0 THEN
				nProcessFeedback := ipStation[nForCounter].P_nErrorCode;
			END_IF
		END_IF
	END_FOR	

	ipMotionSystemApplication.Execute();
	

	(*
	StateComplete();	// <- nothing will happen since there's no state defined after Execute,
						//    instead Execute can only be left by the Operator pressing the Abort-Button.
	*)
END_METHOD

METHOD HoldOnError : BOOL
VAR_INPUT
END_VAR



CASE nStateSequence OF
	0: 		
		IF ipMotionSystemApplication <> 0 THEN
			nStateSequence := 10;
		END_IF

	10:	
		IF nProcessFeedback = 0 THEN
			nStateSequence := 99;
		END_IF

	100:
		StateComplete();
END_CASE
END_METHOD

PROPERTY P_bErrorQuit : BOOL
SET
bErrorQuit := P_bErrorQuit;
END_SET
END_PROPERTY

PROPERTY P_nProcessFeedback : UDINT
GET
P_nProcessFeedback := nProcessFeedback;
END_GET
END_PROPERTY

METHOD PRIVATE Prepared
VAR_INPUT
END_VAR


	nTestCounter_Prepared := nTestCounter_Prepared +1;
	
	
	(*
		Prepared: 
		- all movers active (flying)
		- all movers in home position
	
	*)
END_METHOD

{attribute 'object_name' := 'Preparing'}
METHOD PRIVATE Preparing
CASE nStateSequence OF
	0: 		

		FOR nForCounter:=1 TO nStationCount DO
			IF ipStation[nForCounter] <> 0 THEN
				ipStation[nForCounter].Processing(i_nMachineState:=1);				
				IF ipStation[nForCounter].P_nErrorCode > 0 THEN
					nProcessFeedback := ipStation[nForCounter].P_nErrorCode;
				END_IF
			END_IF
		END_FOR	
		
		
		IF ipMotionSystemApplication.Starting() THEN
			nStateSequence := 100;
		END_IF

	100:
		StateComplete();
END_CASE
END_METHOD

{attribute 'object_name' := 'Resetting'}
METHOD PRIVATE Resetting
CASE nStateSequence OF
	0: 
		
		IF ipMotionSystemApplication.Resetting() THEN
			nStateSequence := 10;
		END_IF

	10:
		IF  ipStation[1].ClearList()
		AND ipStation[2].ClearList()
		AND ipStation[3].ClearList() 
		THEN
			nStateSequence := 100;
		END_IF
		
		
	100:
		StateComplete();
END_CASE
END_METHOD

{attribute 'object_name' := 'StartUp'}
METHOD PRIVATE StartUp
VAR
	nForCounter : UDINT;
END_VAR
CASE nStateSequence OF


	0: 	// XPlanar- or XTS-System?
		{IF defined (XPlanar)}	
		fbMotionSystem.std := THIS^.fbXPlanarSystem;
		{ELSIF defined (XTS)}
		fbMotionSystem.std := THIS^.fbXtsSystem;
		{END_IF}
		nStateSequence := 1;
		
	1:  // Mover assignment 
		FOR nForCounter := 1 TO moverCount DO
			{IF defined (XPlanar)}	
			fbMover[nForCounter].std := THIS^.fbXPlanarMover[nForCounter];
			{ELSIF defined (XTS)}
			fbMover[nForCounter].std := THIS^.fbXtsMover[nForCounter];
			{END_IF}
		END_FOR	
		nStateSequence := 2;
	
	2:	// Writing motion system to global motion system interface
		ipMotionSystemApplication := THIS^.fbMotionSystem;
		nStateSequence := 3;
			
	3:  // Writing movers to global mover interface
		FOR nForCounter := 1 TO moverCount DO
			ipMoverApplication[nForCounter] := THIS^.fbMover[nForCounter];
			THIS^.fbMover[nForCounter].P_nMoverIndex := UDINT_TO_INT(nForCounter); 
		END_FOR	
		nStateSequence := 4;

	4:  // Assigning Track-Interfaces
		ipTrack[1] := THIS^.fbTrackSegment01;
		ipTrack[2] := THIS^.fbTrackSegment02;
		ipTrack[3] := THIS^.fbTrackSegment03;	
		nStateSequence := 5;	
					
	5:  // Assigning Station-Interfaces
		ipStation[1] := THIS^.fbStation_01_Process;
        ipStation[2] := THIS^.fbStation_02_Process;		
        ipStation[3] := THIS^.fbStation_03_Process;			
		ipStation[4] := THIS^.fbStation_04_Switch;
		ipStation[5] := THIS^.fbStation_05_Switch;	
	
		bInterfaceAssignmentDone := TRUE;
		nStateSequence := 10;
	
	
	10: // Calling Application-Startup-Procedure	
		IF ipMotionSystemApplication.Startup() THEN
			nStateSequence := 100;
		END_IF
	

	100: // Start-up done
		StateComplete();
END_CASE
END_METHOD

{attribute 'object_name' := 'StateComplete'}
METHOD PRIVATE StateComplete

	nTestCounter_StateComplete := nTestCounter_StateComplete + 1;

	nStateSequence := 0;
	
	//the actual state is completed
	fbStateManager.StateComplete();
END_METHOD

{attribute 'object_name' := 'Stopped'}
METHOD PRIVATE Stopped

	nTestCounter_Stopped := nTestCounter_Stopped + 1;


	(*
	
		Stopped: 
		- Production finished
		- …
		
	*)
END_METHOD

PROPERTY PUBLIC XCommand : E_XMotion_Command
SET
  eXCommand := XCommand;
END_SET
END_PROPERTY

PROPERTY PUBLIC XMotionStatus : E_XMotion_Status
GET
   XMotionStatus := eXStatus;
END_GET
END_PROPERTY

PROPERTY XSequenceStates : ST_XMotionStatemachineStates
GET
XSequenceStates := stSequenceStates;
END_GET
END_PROPERTY

END_FUNCTION_BLOCK

// ---- 2_Application/Machine/FB_MotionSystem.TcPOU
FUNCTION_BLOCK FB_MotionSystem IMPLEMENTS I_MotionSystemApplication
VAR_INPUT
END_VAR
VAR_OUTPUT
END_VAR
VAR
	
	ipMotionSystem			: I_MotionSystem;
	stMoverDetectionInfos   : ST_TcIoMoverDetectionInfos;

	bMoverError	: BOOL;	
	
	// Dynamic limitations
	fVelo           		: LREAL := 250.0;
	fAccel    				: LREAL := 3000.0;
	fJerk            		: LREAL := 30000.0;

	// Sequences
	nStartupSequence 		: UDINT;
	nAbortingSequence 		: UDINT;
	nStartingSequence 		: UDINT;
	nResettingSequence 		: UDINT;
	nExecutingSequence 		: UDINT;	
	
	// Helper
	bDone 					: BOOL;
	nForCounter 			: UDINT;	

	// Temp
	tonDelay		: TON;
	
	
END_VAR

METHOD Aborting : BOOL
VAR

END_VAR
CASE nAbortingSequence OF 

	0: //Idle	
		nAbortingSequence := 10; 	

	10: // Sending "Halt" to all movers for immediate stop 
		IF ipMotionSystem.HaltSystem() THEN
			nAbortingSequence := nAbortingSequence +1;
		ELSE 
			nAbortingSequence := nAbortingSequence +5;	
		END_IF
		
	11: IF ipMotionSystem.P_HaltSystem.Done THEN
			nAbortingSequence := 20;
		ELSIF ipMotionSystem.P_HaltSystem.Error THEN
			;
		END_IF	
	
		
	20:// All movers leave their track
		IF ipMotionSystem.LeaveTrack() THEN
			nAbortingSequence := 21;
		ELSE
			nAbortingSequence := nAbortingSequence +5;
		END_IF
	
	21: IF ipMotionSystem.P_LeaveTrack.Done THEN
			nAbortingSequence := 30;
		ELSIF ipMotionSystem.P_LeaveTrack.Error THEN
			;
		END_IF
		
		
	30: // Removing all movers from the group
		IF ipMotionSystem.RemoveMoversFromGroup() THEN
			nAbortingSequence := 31;
		END_IF

	31: IF ipMotionSystem.P_RemoveMoversFromGroup.Done THEN
			nAbortingSequence := 40;
		END_IF		


	40: // Disable all movers	
		IF ipMotionSystem.DisableMovers() THEN
			nAbortingSequence := 41;
		ELSE
			nAbortingSequence := nAbortingSequence +5;
		END_IF

	41: IF ipMotionSystem.P_DisableMovers.Done THEN
			nAbortingSequence := 50;
		END_IF

		
	50: // Disable group
		IF ipMotionSystem.DisableGroup() THEN
			nAbortingSequence := 51;
		END_IF

	51: IF ipMotionSystem.P_DisableGroup.Done THEN
			nAbortingSequence := 60;
		END_IF		
		
	60: // Remove Environment from Group
		IF ipMotionSystem.RemoveEnvironmentFromGroup() THEN
			nAbortingSequence := 61;
		END_IF	
		
	61: IF ipMotionSystem.P_RemoveEnviromentFromGroup.Done THEN
			nAbortingSequence := 70;
		END_IF		

	70: // Diable all tracks	
		FOR nForCounter := 1 TO trackCount DO
			ipTrack[nForCounter].std.Disable();
		END_FOR
		nAbortingSequence := 80;
	
	80:	nAbortingSequence := 100;
		ipMotionSystemApplication.P_bMoverError := FALSE; //  Only for testing

	100: // Reset of all sequences / Aborting done
		nAbortingSequence  := 0;
		nResettingSequence := 0;
		nStartingSequence  := 0;
		nExecutingSequence := 0;
		          Aborting := TRUE;
 
END_CASE
END_METHOD

METHOD Cycle : BOOL
VAR_INPUT
END_VAR



VAR_INST
	nMoverIndex	: UDINT;

END_VAR
bMoverError := FALSE;

// Scanning for mover error e.g. Following Error
FOR nMoverIndex:=1 TO moverCount DO	
	IF ipMoverApplication[nMoverIndex] <> 0 THEN
		IF ipMoverApplication[nMoverIndex].std.P_State = MC_PLANAR_STATE.Error THEN
			bMoverError := TRUE;	
		END_IF
	END_IF
END_FOR
END_METHOD

METHOD Execute : UDINT




VAR_INST
	


END_VAR
;
END_METHOD

METHOD INTERNAL MoverRecovery : BOOL
VAR_INPUT
	bReset	: BOOL;
END_VAR



VAR_INST

	// Dynamic limitations
	fVeloRec           				: LREAL := 250.0;
	fAccelRec    					: LREAL := 3000.0;
	fJerkRec            			: LREAL := 30000.0;

	idx								: UDINT;	
	nTestCounter					: UDINT;
	nStateMoverRecovery				: INT;	
	bAllMoversDone					: BOOL;
	nForCounter						: UDINT;
	bStillBusy						: BOOL;
	nInitPositionToMoveTo			: UDINT;
	bAllMoversAtInitPosition		: BOOL;
	nInitPositionIndex	  			: UDINT;
	nMoverIndex			  			: UDINT;
	nMoversToInitPositionFound		: UDINT;
	nMoverToJoinTrack				: UDINT;
	nMoverToInitPosition			: UDINT;
	bTryMoveX						: BOOL;
	bTryMoveY						: BOOL;
	nCounterMoverToMove				: INT;	
	
	fInitialMoverPosition			: ARRAY [1..MaxMovers,1..2] OF LREAL;
	bMoverSortedAlready				: ARRAY [1..MaxMovers] OF BOOL;
	bMoverSkipInitPosition			: ARRAY [1..MaxMovers] OF BOOL;
	bMoverToInitPosition			: ARRAY [1..MaxMovers] OF BOOL;
	bMoverAtInitPosition			: ARRAY [1..MaxMovers] OF BOOL;
	bMoverBlockedByMove				: ARRAY [1..MaxMovers] OF BOOL;
	bInitPositionBlockedByMove		: ARRAY [1..MaxMovers] OF BOOL;	
	bInitialMoverPositionDone		: ARRAY [1..MaxMovers] OF BOOL;
	nMoverOnTheWayToInitPosition	: ARRAY [1..MaxMovers] OF UDINT;
	fMoverDistanceToInitialPosition	: ARRAY [1..MaxMovers] OF LREAL;
	fShortestDistance				: ARRAY [1..MaxMovers] OF LREAL;
	nClosestMoverToInitPosition		: ARRAY [1..MaxMovers] OF UDINT;
	nInitPositionMoverTable			: ARRAY [1..MaxMovers] OF UDINT;
	nMoverRecoveryPosition			: ARRAY [1..MaxMovers] OF UDINT;
	nJoinTrack						: ARRAY [1..MaxMovers] OF UDINT;	

	targetPos            	 		: PositionXYC;
    currentPos			     		: PositionXYC;
	nCmdReturnError					: UDINT;
	
	
//-----------------first Track run

	fTrackLengthTrack1  	: LREAL;
	fTrackLengthTrack2  	: LREAL;	
	fTrackLengthTrack3  	: LREAL;	
	
	bInitRunFlag			: BOOL;
	bInitRunDone			: BOOL;
	bOneMoverMoving			: BOOL;
	bAllMoversStandingStill	: BOOL;
	bMoversQueuing			: BOOL;
	
	TimerWaitForMovement	: TON;	
	
	
	nState 					: INT;	
	nStateInit				: INT;
	
	
	fbInitList				: FB_List;

	fPositionOnTrack			: LREAL;
	nStationIndex				: UINT;
	nNextStationTrackIndex 		: UINT;
	fNextStationWaitingPosition	: LREAL;
	nTrackIndex					: UDINT;
	nNextStationIndex			: UDINT;
	bFirstMoverIn				: BOOL;
	ClearTrig					: R_TRIG;
	fMoverPosition				: LREAL;
	fMoverVelocity				: LREAL;
	fMoverAcceleration			: LREAL;
	fMoverJerk					: LREAL;
	strInfo						: STRING;
	
	fMoverSpace					: LREAL;
	fWaitingPositionStation01	: LREAL;
	fWaitingPositionStation02	: LREAL;	
	fWaitingPositionStation03	: LREAL;	
	fWaitingPositionStation04	: LREAL;	
	fWaitingPositionStation05b	: LREAL;	
	fWaitingPositionStation05c	: LREAL;
	
	stMoveParameters 	: ST_MoveOnTrackOptions; 
	strInfoHistory		: ARRAY[0..10] OF STRING;
	
	nResult				: DINT;
	sMessage			: STRING;
	
	
END_VAR
IF bReset THEN
	nStateMoverRecovery := 0;
END_IF



CASE nStateMoverRecovery OF

	
	(***************************************************************************************)
	(* Mover Recovery Part1: Separating all movers and move each of them to a corner point *)
	(*                       specified by fInitialMoverPosition                            *)
	(***************************************************************************************)                                  

	0:		// Starting mover recovery
				  MoverRecovery := FALSE;
			nStateMoverRecovery := 10;
	
			
	10:		// Setting initial-points for mover sorting				
			fInitialMoverPosition[1,1] := 120.0;
			fInitialMoverPosition[1,2] := 120.0;	
			
			fInitialMoverPosition[2,1] := 120.0;
			fInitialMoverPosition[2,2] := 600.0;		
			
			fInitialMoverPosition[3,1] := 840.0;
			fInitialMoverPosition[3,2] := 600.0;		
		
			fInitialMoverPosition[4,1] := 840.0;
			fInitialMoverPosition[4,2] := 120.0;
	
			fbInitList.ClearList();
			
			nStateMoverRecovery := 100;
			
		
	100: // -> All movers to their initial position
				
			// Resetting all flags 
			FOR idx:=1 TO moverCount DO
						bMoverToInitPosition[idx] := FALSE;
					  bMoverSkipInitPosition[idx] := FALSE;
						 bMoverSortedAlready[idx] := FALSE;
						bMoverAtInitPosition[idx] := FALSE;
				  bInitPositionBlockedByMove[idx] := FALSE;
					 nInitPositionMoverTable[idx] := 0;
				nMoverOnTheWayToInitPosition[idx] := 0;
			END_FOR		
			nStateMoverRecovery:= 110;
			
			
	110:  // -> Figuring out which mover needs to go to which init-position
			
			// Cleaning working registers
				 nInitPositionToMoveTo := 0;	
			nMoversToInitPositionFound := 0;
			FOR idx:=1 TO moverCount DO
				nClosestMoverToInitPosition[idx] := 0;
						bMoverSortedAlready[idx] := FALSE;
						  fShortestDistance[idx] := 1.7976931348623158E+308;		 
			END_FOR
			
			// Release mover blocking after movement
			FOR idx:=1 TO moverCount DO
				IF NOT ipMoverApplication[idx].std.P_MoveToPosition.Busy THEN
						   bMoverBlockedByMove[idx] := FALSE;
				END_IF
			END_FOR
				
			// Finding closest mover to each init-position
			FOR nInitPositionIndex:=1 TO moverCount DO
				IF bInitPositionBlockedByMove[nInitPositionIndex] = FALSE THEN
					FOR nMoverIndex:=1 TO moverCount DO  
						IF  NOT     bMoverToInitPosition[nMoverIndex]
						AND NOT     bMoverAtInitPosition[nMoverIndex]
						AND NOT      bMoverSortedAlready[nMoverIndex]
						AND NOT      bMoverBlockedByMove[nMoverIndex]
						AND NOT   bMoverSkipInitPosition[nMoverIndex]
						AND nMoverOnTheWayToInitPosition[nMoverIndex]=0				
						THEN
							currentPos.SetValuesXYC(ipMoverApplication[nMoverIndex].std.P_SetPosition.x, ipMoverApplication[nMoverIndex].std.P_SetPosition.y, ipMoverApplication[nMoverIndex].std.P_SetPosition.c);
							fMoverDistanceToInitialPosition[nMoverIndex] := SQRT((currentPos.x - fInitialMoverPosition[nInitPositionIndex,1]) * (currentPos.x - fInitialMoverPosition[nInitPositionIndex,1]) + (currentPos.y - fInitialMoverPosition[nInitPositionIndex,2]) * (currentPos.y - fInitialMoverPosition[nInitPositionIndex,2])); 
					
							IF fMoverDistanceToInitialPosition[nMoverIndex] < fShortestDistance[nInitPositionIndex] THEN
										  fShortestDistance[nInitPositionIndex] := fMoverDistanceToInitialPosition[nMoverIndex];
								nClosestMoverToInitPosition[nInitPositionIndex] := nMoverIndex;	
													 nMoversToInitPositionFound := nMoversToInitPositionFound + 1;
							END_IF
						END_IF
					END_FOR
					IF nClosestMoverToInitPosition[nInitPositionIndex] > 0 THEN
						bMoverSortedAlready[nClosestMoverToInitPosition[nInitPositionIndex]] := TRUE;
					END_IF
				END_IF	
			END_FOR
					
			// Building the table which defines which mover must go to which init-position
			nCounterMoverToMove := 0;
			FOR nInitPositionIndex:=1 TO moverCount DO 
				nInitPositionMoverTable[nInitPositionIndex] := nClosestMoverToInitPosition[nInitPositionIndex];
				IF nInitPositionMoverTable[nInitPositionIndex] <> 0 THEN
					nCounterMoverToMove := nCounterMoverToMove +1;
				END_IF
			END_FOR
			
			IF nCounterMoverToMove > 0 THEN
				nStateMoverRecovery:= 120;
			ELSE
				// Skipping release
				FOR idx:=1 TO moverCount DO
					bMoverSkipInitPosition[idx] := FALSE;
				END_FOR	
			END_IF
				
		
	120:  // Sending all movers to their init-positions
			nInitPositionToMoveTo := nInitPositionToMoveTo + 1;
			
			IF nInitPositionToMoveTo <= moverCount THEN
				IF nInitPositionMoverTable[nInitPositionToMoveTo] > 0 THEN
					nMoverToInitPosition := nInitPositionMoverTable[nInitPositionToMoveTo]; 
					nMoverRecoveryPosition[nMoverToInitPosition] := nInitPositionToMoveTo;
					nStateMoverRecovery := 130;
				END_IF
			ELSE
				nStateMoverRecovery := 121; 
			END_IF
				
			
	121:  // Waiting for all movers standing still
			bStillBusy := FALSE;
			FOR idx:=1 TO moverCount DO
				IF ipMoverApplication[idx].std.P_MoveToPosition.Busy THEN
					bStillBusy := TRUE;
				ELSE
					IF bMoverToInitPosition[idx] THEN 
								bMoverToInitPosition[idx] := FALSE;
								bMoverAtInitPosition[idx] := TRUE;					
						nMoverOnTheWayToInitPosition[idx] := 0;
					END_IF				
				END_IF
			END_FOR
		
			IF NOT bStillBusy THEN
				nStateMoverRecovery := 122; 
			END_IF
				
			
	122:  // Checking if all movers at their init-position 
			bAllMoversAtInitPosition := TRUE;
			FOR idx:=1 TO moverCount DO	
				IF NOT bMoverAtInitPosition[idx] THEN
					bAllMoversAtInitPosition := FALSE;
				END_IF
			END_FOR
			
			IF bAllMoversAtInitPosition THEN
				nStateMoverRecovery := 150;   // All movers are now at their init-position.
			ELSE
				nStateMoverRecovery := 110;	// Try another round to move previously blocked movers.
			END_IF		
			
		
	130: 	// Move a mover to its init-position
			IF NOT ipMoverApplication[nMoverToInitPosition].std.P_MoveToPosition.Busy THEN	
				targetPos.SetValuesXYC(fInitialMoverPosition[nInitPositionToMoveTo,1],fInitialMoverPosition[nInitPositionToMoveTo,2],0);
				IF ipMoverApplication[nMoverToInitPosition].std.MoveToPosition('',targetPos,fVeloRec,fAccelRec,fAccelRec,fJerkRec) THEN
					nStateMoverRecovery:= 131;
				END_IF
			END_IF
						
		
	131:	// ...decide accoding to command return
			nCmdReturnError := ipMoverApplication[nMoverToInitPosition].std.P_MoveToPosition.ErrorID;
	
			IF ipMoverApplication[nMoverToInitPosition].std.P_MoveToPosition.Active  	
			OR ipMoverApplication[nMoverToInitPosition].std.P_MoveToPosition.Error 
			OR ipMoverApplication[nMoverToInitPosition].std.P_MoveToPosition.Done
			THEN		
				IF nCmdReturnError = 0 THEN 
							 bMoverBlockedByMove[nMoverToInitPosition] := TRUE;
					 bInitPositionBlockedByMove[nInitPositionToMoveTo] := TRUE;
							bMoverToInitPosition[nMoverToInitPosition] := TRUE;
					nMoverOnTheWayToInitPosition[nMoverToInitPosition] := nInitPositionToMoveTo;
						 
					FOR idx:=1 TO moverCount DO	
						bMoverSkipInitPosition[idx] := FALSE;
					END_FOR						
					nStateMoverRecovery := 140;	
			
				ELSIF nCmdReturnError = 33158 THEN   // 33158 = Collision
					
					IF NOT bTryMoveX THEN
						nStateMoverRecovery:= 132;
					ELSIF NOT bTryMoveY THEN
						nStateMoverRecovery:= 134;
					ELSE	
						nMoverOnTheWayToInitPosition[nMoverToInitPosition] := 0;
						nStateMoverRecovery:= 140;
					END_IF
				END_IF			
			END_IF
	
		
	132: 	// try x-direction
			IF NOT ipMoverApplication[nMoverToInitPosition].std.P_MoveToPosition.Busy THEN		
				bTryMoveX := TRUE;
				currentPos.SetValuesXYC(ipMoverApplication[nMoverToInitPosition].std.P_SetPosition.x, ipMoverApplication[nMoverToInitPosition].std.P_SetPosition.y, ipMoverApplication[nMoverToInitPosition].std.P_SetPosition.c);
				targetPos.SetValuesXYC(fInitialMoverPosition[nInitPositionToMoveTo,1],currentPos.y,0);
				ipMoverApplication[nMoverToInitPosition].std.MoveToPosition('',targetPos,fVeloRec,fAccelRec,fAccelRec,fJerkRec);
				
				nStateMoverRecovery:= 133;
			END_IF
			
	133:	// ...decide accoding to command return
			nCmdReturnError := ipMoverApplication[nMoverToInitPosition].std.P_MoveToPosition.ErrorID;
	
			IF ipMoverApplication[nMoverToInitPosition].std.P_MoveToPosition.Active
			OR ipMoverApplication[nMoverToInitPosition].std.P_MoveToPosition.Error
			OR ipMoverApplication[nMoverToInitPosition].std.P_MoveToPosition.Done
			THEN	
			
				IF nCmdReturnError = 0 THEN
							 bMoverBlockedByMove[nMoverToInitPosition] := TRUE;
					nMoverOnTheWayToInitPosition[nMoverToInitPosition] := nInitPositionToMoveTo;
					
					nStateMoverRecovery:= 130;
					
				ELSIF nCmdReturnError = 33158 THEN   // 33158 = Collision	
					bMoverSkipInitPosition[nMoverToInitPosition] := TRUE;
					
					nStateMoverRecovery:= 130;
				END_IF	
			END_IF
				
	134: 	// try y-direction
			IF NOT ipMoverApplication[nMoverToInitPosition].std.P_MoveToPosition.Busy THEN
				bTryMoveY := TRUE;
				currentPos.SetValuesXYC(ipMoverApplication[nMoverToInitPosition].std.P_SetPosition.x, ipMoverApplication[nMoverToInitPosition].std.P_SetPosition.y, ipMoverApplication[nMoverToInitPosition].std.P_SetPosition.c);
				targetPos.SetValuesXYC(currentPos.x ,fInitialMoverPosition[nInitPositionToMoveTo,2],0);
				ipMoverApplication[nMoverToInitPosition].std.MoveToPosition('',targetPos,fVeloRec,fAccelRec, fAccelRec,fJerkRec);
	
				nStateMoverRecovery:= 135;
			END_IF
			
	135:	// ...decide accoding to command return
			nCmdReturnError := ipMoverApplication[nMoverToInitPosition].std.P_MoveToPosition.ErrorID;
			
			IF ipMoverApplication[nMoverToInitPosition].std.P_MoveToPosition.Active
			OR ipMoverApplication[nMoverToInitPosition].std.P_MoveToPosition.Error
			OR ipMoverApplication[nMoverToInitPosition].std.P_MoveToPosition.Done
			THEN					
				IF nCmdReturnError = 0 THEN
							 bMoverBlockedByMove[nMoverToInitPosition] := TRUE;
					nMoverOnTheWayToInitPosition[nMoverToInitPosition] := nInitPositionToMoveTo;
					
					nStateMoverRecovery:= 130;
					
				ELSIF nCmdReturnError = 33158 THEN   // 33158 = Collision			
					bMoverSkipInitPosition[nMoverToInitPosition] := TRUE;
					
					nStateMoverRecovery:= 130;
				END_IF
			END_IF
			
	140:
		// Clean flags for next mover to be moved				
		bTryMoveX := FALSE;
		bTryMoveY := FALSE;	
		nStateMoverRecovery:= 120;
		
		
	150:

		bDone := TRUE;
		FOR nForCounter := 1 TO moverCount DO
			bDone := bDone AND ipMoverApplication[nForCounter].std.P_MoveToPosition.Done;
		END_FOR
		
		IF bDone THEN 
			nStateMoverRecovery := 139;
		END_IF
		
		// Clean flags for next mover to be moved				
			bTryMoveX := FALSE;
			bTryMoveY := FALSE;	
			nStateMoverRecovery:= 200;
			

	
			
	(***************************************************************************************)
	(* Mover Recovery Part2: All movers join the outer-track							   *)
	(***************************************************************************************)  	
					
			
	200:	// All movers go on track
			FOR nForCounter := 1 TO moverCount DO
				IF ipMoverApplication[nForCounter].std.P_SetPosition.x > 480.0 THEN
					nJoinTrack[nForCounter] := 3;	
				ELSE
					nJoinTrack[nForCounter] := 1;	
				END_IF
			END_FOR
			nStateMoverRecovery := 201;	
				
	201:	IF nMoverToJoinTrack < moverCount THEN
				nMoverToJoinTrack := nMoverToJoinTrack +1;
				nStateMoverRecovery := nStateMoverRecovery +1;
			ELSE
				nMoverToJoinTrack := 0;
				nStateMoverRecovery := nStateMoverRecovery + 2; 
			END_IF
				
	202:	IF ipMoverApplication[nMoverToJoinTrack].std.JoinTrack('',ipTrack[nJoinTrack[nMoverToJoinTrack]].std, fVeloRec, fAccelRec, fJerkRec) THEN
				ipMoverApplication[nMoverToJoinTrack].P_nTrackId := nJoinTrack[nMoverToJoinTrack];
				nStateMoverRecovery := nStateMoverRecovery -1;
			END_IF
			
	203:	bDone := TRUE;
			FOR nForCounter := 1 TO moverCount DO
				bDone := bDone AND ipMoverApplication[nForCounter].std.P_JoinTrack.Done;
			END_FOR
			
			IF bDone THEN
				nStateMoverRecovery := 210;
			END_IF
		
	210:  // Wait for all movers on-track
			bDone := TRUE;
			FOR nForCounter := 1 TO moverCount DO
				bDone := bDone AND ipMoverApplication[nForCounter].std.P_JoinTrack.Done;
			END_FOR
			IF bDone THEN
				nStateMoverRecovery := 220;
			END_IF
	
			
	
	(***************************************************************************************)
	(* Mover Recovery Part3: Adding all movers to the Initialization-List and sort them    *)
	(*                       ascending.                              				       *)
	(***************************************************************************************)  			
				
			
	220:	// Adding all movers to the Initialization-List
			FOR nForCounter := 1 TO moverCount DO
				fbInitList.AddMover(ipMoverApplication[nForCounter].std);
			END_FOR				
			nStateMoverRecovery := 230;
			
			
	230: 	// Adding Track-Order to the Initialization-List for Sorting-Order
			IF fbInitList.AddTrack(ipTrack[1].std) > 0 THEN
				nStateMoverRecovery := 231;
			ELSE
				 nResult := fbInitList.P_nResult;
				sMessage := fbInitList.P_sMessage;	
			END_IF
			
	231: 	IF fbInitList.AddTrack(ipTrack[3].std) > 0 THEN
				nStateMoverRecovery := 232;
			ELSE
				 nResult := fbInitList.P_nResult;
				sMessage := fbInitList.P_sMessage;	
			END_IF			
						
 	232:	nStateMoverRecovery := 238;
		
				
	238:	// Sorting all movers 
			 nResult := fbInitList.SortList();
			sMessage := fbInitList.P_sMessage;
			
			IF nResult > 0 THEN
				// Sorting succesful - will return the number of movers sorted e.g. 4
				nStateMoverRecovery:= 240;
			ELSIF nResult = 0 THEN
				;// Sorting 
			ELSIF nResult < 0 THEN
				// sorting Error - Check error code and error message
				nStateMoverRecovery:= 239;
			END_IF
	
	240:	nStateMoverRecovery:= 250;			
	

	
	(***************************************************************************************)
	(* Mover Recovery Part4: Initialization-Run                                            *)
	(*						 - Sending/Adding each mover to its next closest station       *)
	(*						 - From there on each station takes care of the init-run       *)
	(* 						 - Movers will queu in in front of station 01 				   *)
	(***************************************************************************************)  

	250: // Init all variables 
					bOneMoverMoving := FALSE;
			bAllMoversStandingStill := FALSE;
					   bInitRunDone := FALSE;
	
				   nStateMoverRecovery := 300;
	
	300: // Check for next Mover
		IF fbInitList.P_FirstInList <> 0 THEN
				 nMoverIndex := fbInitList.P_FirstInList.P_Id;
				 nTrackIndex := ipMoverApplication[nMoverIndex].P_nTrackId;
			fPositionOnTrack := ipMoverApplication[nMoverIndex].std.P_SetOnTrack.SetPos;
			
			bFirstMoverIn := TRUE;
				   nStateMoverRecovery := 310;
		ELSE
			IF bFirstMoverIn THEN
				nStateMoverRecovery := 305;
			ELSE
				// Init-Run completed
				bInitRunFlag := FALSE;
				nStateMoverRecovery := 500;	
			END_IF
		END_IF
			
		
	305: // Wait till at least one mover started moving, or timeout if no movement at all.
		bOneMoverMoving := FALSE;
		FOR idx:=1 TO moverCount DO	
			IF ABS(ipMoverApplication[idx].std.P_SetVelocity.x) > 0.1
			OR ABS(ipMoverApplication[idx].std.P_SetVelocity.y) > 0.1
			THEN
				bOneMoverMoving := TRUE;
			END_IF
		END_FOR		
	
		TimerWaitForMovement(IN:=TRUE, PT:=T#2S);
		
		IF bOneMoverMoving 
		OR TimerWaitForMovement.Q 
		THEN
			TimerWaitForMovement(IN:=FALSE);
			nStateMoverRecovery := 306;			
		END_IF
			
		
	306: // Wait till all movers are standing still	
		bAllMoversStandingStill := TRUE;
		FOR idx:=1 TO moverCount DO	
			IF ABS(ipMoverApplication[idx].std.P_SetVelocity.x) > 0.001
			OR ABS(ipMoverApplication[idx].std.P_SetVelocity.y) > 0.001
			THEN
				bAllMoversStandingStill := FALSE;
			END_IF
		END_FOR
	
		IF bAllMoversStandingStill THEN
			bMoversQueuing := TRUE; 
			FOR idx:=2 TO moverCount DO
				IF NOT (ipMoverApplication[idx].std.P_MoveOnTrack.Busy OR ipMoverApplication[idx].std.P_MoveOnTrack.done) THEN
					bMoversQueuing := FALSE;	
				END_IF
			END_FOR
		ELSE
			bMoversQueuing := FALSE;
		END_IF
		
		IF bMoversQueuing THEN
			       bInitRunDone := TRUE;
			nStateMoverRecovery := 500;			
		END_IF
	
		
	310: // Figuring out the next station the mover has to travel to:
		fMoverSpace := 155.0 + 5.0;
	
		fWaitingPositionStation01	:= ipTrack[1].P_TrackLength/2.0 - fMoverSpace;	
		fWaitingPositionStation02	:= ipTrack[2].P_TrackLength/2.0 - fMoverSpace;	
		fWaitingPositionStation03	:= ipTrack[3].P_TrackLength/2.0 - fMoverSpace;
		fWaitingPositionStation04	:= ipTrack[1].P_TrackLength - fMoverSpace;	
		fWaitingPositionStation05b	:= ipTrack[3].P_TrackLength - fMoverSpace;	
		fWaitingPositionStation05c	:= ipTrack[2].P_TrackLength - fMoverSpace;	
	
		CASE nTrackIndex OF		
		1:	// Mover on Track01 / Station01
			IF fPositionOnTrack <= fWaitingPositionStation01 THEN
				nNextStationIndex := 1;
			ELSE
				nNextStationIndex := 4;
			END_IF	
	
		2:	// Mover on Track02 / Station02
			IF fPositionOnTrack <= fWaitingPositionStation02 THEN
				nNextStationIndex := 2;
			ELSE
				nNextStationIndex := 5;
			END_IF			
		
		3:	// Mover on Track03 / Station 03
			IF fPositionOnTrack <= fWaitingPositionStation03 THEN
				nNextStationIndex := 3;
			ELSE
				nNextStationIndex := 5;
			END_IF			
		END_CASE
		
		nStateMoverRecovery := 320;
			
			
	320: // Calculating the position the mover has to move to next:
		nNextStationTrackIndex := 0;
		
		CASE nNextStationIndex OF
			1:	nNextStationTrackIndex      := 1;
				fNextStationWaitingPosition	:= fWaitingPositionStation01;	
			
			2:	nNextStationTrackIndex      := 2;
				fNextStationWaitingPosition	:= fWaitingPositionStation02;			
			
			3:	nNextStationTrackIndex      := 3;
				fNextStationWaitingPosition	:= fWaitingPositionStation03;			
			
			4:	nNextStationTrackIndex      := 1;
				fNextStationWaitingPosition	:= fWaitingPositionStation04;				
				
			5:	IF nTrackIndex = 2 THEN
					nNextStationTrackIndex := 2;
					fNextStationWaitingPosition	:= fWaitingPositionStation05c;	
				ELSIF nTrackIndex = 3 THEN
					nNextStationTrackIndex := 3;
					fNextStationWaitingPosition	:= fWaitingPositionStation05b;	
				END_IF									
		END_CASE
			
		IF nNextStationTrackIndex > 0 THEN
			nStateMoverRecovery := 400;
		END_IF
	
	
